FUNCTION_BLOCK sifb_bfb_inputs
  (* Standard: 61499-2 *)
  (* Version 0.1, 2018-00-07, hpea485, UOA *)
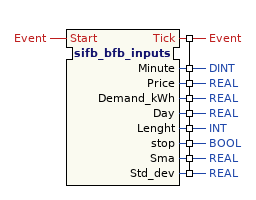
  EVENT_INPUT
    Start;
  END_EVENT
  EVENT_OUTPUT
    Tick WITH Minute, Price, Demand_kWh, Day, Lenght, stop, Sma, Std_dev;
  END_EVENT
  VAR_OUTPUT
    Minute : DINT;
    Price : REAL;
    Demand_kWh : REAL;
    Day : REAL;
    Lenght : INT;
    stop : BOOL;
    Sma : REAL;
    Std_dev : REAL;
  END_VAR
  VAR
    Var : DINT;
  END_VAR
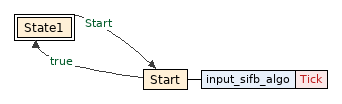
  EC_STATES
    State1;
    Start : input_sifb_algo -> Tick;
  END_STATES
  EC_TRANSITIONS
    Start TO State1 := true;
    State1 TO Start := Start;
  END_TRANSITIONS
  ALGORITHM input_sifb_algo IN C:
//#include "sifb_bfb_inputs.fb.Algorithm1.algo"
//#include "SMA_function.c"
#include <math.h>
static DINT current_minute = 0;
static DINT minute_for_demand = 0;
static DINT lol = 0;

static REAL Sma_tot = 0;
static int j = 1;
static REAL Std_dev;
static int nb_samples;

static int i = 0;
static int l = 8;
static int day = 0;
REAL Sma_forwrd=0;
REAL Sma_backwrd=0;
REAL Std_forwrd_sum = 0;
REAL Std_backwrd_sum = 0;
static bool stop = 0;
#define NUM_HALF_HOURS  48
#define NUM_DAYS        7 //31
me->stop = stop;



static REAL power_demand[1441][NUM_DAYS] = {
	{0,0,0,0,0,0,0},
	{176.7331, 236.0112, 169.5329, 136.7712, 100.643, 134.9339, 135.2902},
	{176.7331, 274.0112, 273.126, 280.6114, 275.0023, 273.324, 274.835},
	{176.7331, 274.0112, 273.126, 280.6114, 275.0023, 273.324, 274.835},
	{176.7331, 274.0112, 273.126, 280.6114, 275.0023, 273.324, 274.835},
	{176.7331, 274.0112, 273.126, 280.6114, 275.0023, 273.324, 274.835},
	{176.7331, 274.0112, 273.126, 280.6114, 275.0023, 273.324, 274.835},
	{176.7331, 274.0112, 273.126, 280.6114, 275.0023, 273.324, 274.835},
	{176.7331, 274.0112, 273.126, 280.6114, 275.0023, 273.324, 274.835},
	{176.7331, 274.0112, 273.126, 280.6114, 275.0023, 273.324, 274.835},
	{176.7331, 274.0112, 273.126, 280.6114, 275.0023, 273.324, 274.835},
	{176.7331, 274.0112, 273.126, 280.6114, 275.0023, 273.324, 274.835},
	{176.7331, 274.0112, 273.126, 280.6114, 275.0023, 273.324, 274.835},
	{176.7331, 274.0112, 273.126, 280.6114, 275.0023, 273.324, 274.835},
	{176.7331, 274.0112, 273.126, 280.6114, 275.0023, 273.324, 274.835},
	{176.7331, 274.0112, 273.126, 280.6114, 275.0023, 273.324, 274.835},
	{176.7331, 274.0112, 273.126, 280.6114, 275.0023, 273.324, 274.835},
	{176.7331, 274.0112, 273.126, 280.6114, 275.0023, 273.324, 274.835},
	{176.7331, 274.0112, 273.126, 280.6114, 275.0023, 273.324, 274.835},
	{176.7331, 274.0112, 273.126, 280.6114, 275.0023, 273.324, 274.835},
	{144.3122, 274.0112, 240.7051, 280.6114, 275.0023, 240.9031, 274.835},
	{144.3122, 209.1694, 240.7051, 280.6114, 242.5814, 240.9031, 242.4141},
	{144.3122, 209.1694, 240.7051, 280.6114, 242.5814, 208.4822, 242.4141},
	{144.3122, 209.1694, 240.7051, 280.6114, 242.5814, 208.4822, 242.4141},
	{144.3122, 175.2002, 240.7051, 212.673, 242.5814, 208.4822, 242.4141},
	{144.3122, 175.2002, 172.7667, 212.673, 208.6122, 208.4822, 174.4757},
	{110.343, 141.231, 138.7975, 212.673, 174.643, 174.513, 140.5065},
	{110.343, 106.231, 138.7975, 212.673, 174.643, 139.513, 140.5065},
	{132.634, 106.231, 103.7975, 142.673, 104.643, 104.513, 105.5065},
	{137.434, 106.231, 103.7975, 107.673, 104.643, 104.513, 105.5065},
	{207.2941, 106.231, 103.7975, 107.673, 104.643, 104.513, 105.5065},
	{207.2941, 106.231, 103.7975, 107.673, 104.643, 104.513, 105.5065},
	{207.2941, 106.231, 103.7975, 107.673, 104.643, 104.513, 105.5065},
	{207.2941, 106.231, 103.7975, 107.673, 104.643, 104.513, 105.5065},
	{207.2941, 106.231, 103.7975, 107.673, 104.643, 104.513, 105.5065},
	{207.2941, 106.231, 103.7975, 107.673, 104.643, 104.513, 105.5065},
	{207.2941, 106.231, 103.7975, 107.673, 103.313, 104.513, 105.5065},
	{202.4941, 106.231, 103.7975, 107.673, 135.7339, 104.513, 105.5065},
	{241.5941, 106.231, 103.7975, 107.673, 135.7339, 104.513, 105.5065},
	{241.5941, 106.231, 103.7975, 107.673, 135.7339, 104.513, 105.5065},
	{241.5941, 106.231, 137.4675, 107.673, 135.7339, 104.513, 105.5065},
	{241.5941, 106.231, 138.7975, 107.673, 135.7339, 136.9339, 105.5065},
	{241.5941, 106.231, 172.7667, 142.673, 135.7339, 136.9339, 105.5065},
	{241.5941, 106.231, 172.7667, 142.673, 135.7339, 136.9339, 105.5065},
	{241.5941, 106.231, 172.7667, 142.673, 135.7339, 136.9339, 105.5065},
	{241.5941, 106.231, 172.7667, 142.673, 135.7339, 136.9339, 105.5065},
	{241.5941, 106.231, 172.7667, 142.673, 135.7339, 136.9339, 105.5065},
	{241.5941, 104.901, 172.7667, 142.673, 135.7339, 136.9339, 105.5065},
	{241.5941, 104.901, 172.7667, 142.673, 135.7339, 136.9339, 105.5065},
	{241.5941, 104.901, 207.3659, 142.673, 135.7339, 136.9339, 105.5065},
	{209.1732, 104.901, 207.3659, 142.673, 135.7339, 136.9339, 105.5065},
	{209.1732, 104.901, 242.3659, 142.673, 135.7339, 136.9339, 105.5065},
	{209.1732, 104.901, 242.3659, 143.373, 135.7339, 136.9339, 105.5065},
	{209.1732, 104.901, 242.3659, 143.373, 135.7339, 136.9339, 139.8065},
	{209.1732, 137.3219, 242.3659, 143.373, 135.7339, 136.9339, 139.8065},
	{140.204, 137.3219, 242.3659, 143.373, 135.7339, 136.9339, 139.8065},
	{140.204, 137.3219, 242.3659, 143.373, 135.7339, 136.9339, 139.1065},
	{140.204, 137.3219, 242.3659, 177.3422, 103.313, 136.9339, 174.1065},
	{140.204, 136.6219, 242.3659, 177.3422, 103.313, 136.9339, 174.1065},
	{140.204, 171.6219, 242.3659, 177.3422, 103.313, 136.9339, 174.1065},
	{140.204, 171.6219, 242.3659, 177.3422, 103.313, 136.9339, 174.1065},
	{140.204, 172.9519, 242.3659, 177.3422, 103.313, 136.9339, 174.1065},
	{140.204, 172.9519, 208.3967, 177.3422, 103.313, 104.513, 174.1065},
	{105.204, 172.9519, 173.3967, 177.3422, 103.313, 140.143, 174.1065},
	{105.204, 207.2519, 173.3967, 177.3422, 137.9822, 140.143, 174.1065},
	{105.204, 207.2519, 173.3967, 142.3422, 104.013, 140.143, 174.1065},
	{105.204, 207.8819, 173.3967, 142.3422, 135.1039, 140.143, 174.1065},
	{105.204, 207.8819, 173.3967, 176.6422, 167.5248, 140.143, 174.1065},
	{105.204, 207.8819, 172.0667, 176.6422, 167.5248, 140.143, 174.1065},
	{105.204, 208.5819, 204.4876, 141.0122, 167.5248, 140.143, 174.1065},
	{105.204, 277.2203, 204.4876, 173.4331, 167.5248, 172.5639, 174.1065},
	{105.204, 277.2203, 170.5184, 173.4331, 167.5248, 172.5639, 174.1065},
	{105.204, 277.2203, 170.5184, 173.4331, 167.5248, 172.5639, 174.1065},
	{105.204, 244.7994, 170.5184, 173.4331, 167.5248, 172.5639, 172.7765},
	{105.204, 244.7994, 170.5184, 173.4331, 166.1948, 172.5639, 205.1974},
	{105.204, 244.7994, 170.5184, 173.4331, 198.6157, 172.5639, 205.1974},
	{105.204, 244.7994, 170.5184, 173.4331, 198.6157, 172.5639, 205.1974},
	{105.204, 244.7994, 204.8184, 173.4331, 198.6157, 172.5639, 205.1974},
	{140.5032, 244.7994, 169.8184, 173.7639, 198.6157, 172.5639, 205.1974},
	{140.5032, 244.7994, 169.8184, 138.1339, 198.6157, 172.5639, 170.1974},
	{140.5032, 244.7994, 169.8184, 170.5548, 198.6157, 204.3548, 135.1974},
	{140.5032, 244.7994, 169.8184, 170.5548, 198.6157, 171.9339, 135.1974},
	{140.5032, 244.7994, 169.8184, 170.5548, 198.6157, 204.3548, 170.8274},
	{140.5032, 244.7994, 169.8184, 205.5548, 198.6157, 204.3548, 135.1974},
	{140.5032, 209.7994, 169.8184, 205.5548, 167.5248, 204.3548, 167.6183},
	{140.5032, 209.7994, 169.8184, 205.5548, 135.1039, 205.0548, 167.6183},
	{141.2032, 209.7994, 137.3975, 205.5548, 135.1039, 237.694, 167.6183},
	{175.1724, 209.7994, 137.3975, 205.5548, 169.0731, 270.1149, 167.6183},
	{175.1724, 209.7994, 137.3975, 205.5548, 169.0731, 235.1149, 167.6183},
	{175.1724, 174.7994, 137.3975, 205.5548, 169.0731, 235.1149, 167.6183},
	{175.1724, 174.7994, 137.3975, 173.1339, 169.0731, 203.324, 167.6183},
	{175.1724, 106.861, 137.3975, 173.1339, 169.0731, 203.324, 167.6183},
	{175.1724, 106.861, 137.3975, 173.1339, 169.0731, 237.9932, 167.6183},
	{175.1724, 141.861, 137.3975, 173.1339, 137.3522, 237.9932, 135.1974},
	{175.1724, 141.861, 137.3975, 173.1339, 171.3214, 237.9932, 135.1974},
	{175.1724, 141.861, 137.3975, 173.1339, 171.3214, 237.9932, 135.1974},
	{175.1724, 141.861, 137.3975, 173.1339, 171.3214, 237.9932, 135.1974},
	{175.1724, 141.861, 137.3975, 173.1339, 171.3214, 237.9932, 135.1974},
	{175.1724, 141.861, 137.3975, 140.713, 171.3214, 237.9932, 135.1974},
	{175.1724, 141.861, 137.3975, 140.713, 171.3214, 237.9932, 135.1974},
	{175.1724, 141.861, 137.3975, 140.713, 171.3214, 237.9932, 134.5674},
	{171.7024, 141.861, 137.3975, 140.713, 171.3214, 237.9932, 166.9883},
	{171.7024, 175.8302, 102.3975, 140.713, 171.3214, 237.9932, 166.9883},
	{137.7332, 175.8302, 102.3975, 140.713, 171.3214, 205.5723, 166.9883},
	{137.7332, 208.2511, 102.3975, 140.713, 171.3214, 205.5723, 166.9883},
	{176.8332, 208.2511, 102.3975, 140.713, 171.3214, 173.1514, 134.5674},
	{176.8332, 208.2511, 102.3975, 140.713, 171.3214, 173.1514, 134.5674},
	{172.0332, 208.2511, 102.3975, 140.713, 171.3214, 173.1514, 134.5674},
	{176.1332, 208.2511, 102.3975, 140.713, 171.3214, 139.1822, 134.5674},
	{211.1332, 208.2511, 102.3975, 105.713, 171.3214, 139.1822, 134.5674},
	{246.1332, 208.2511, 102.3975, 105.713, 137.3522, 139.1822, 134.5674},
	{212.164, 208.2511, 102.3975, 105.713, 137.3522, 171.6031, 134.5674},
	{212.164, 208.2511, 136.3667, 106.343, 137.3522, 171.6031, 134.5674},
	{210.4785, 208.2511, 136.3667, 102.972, 135.6667, 169.9176, 134.5674},
	{210.4785, 208.2511, 100.712, 102.972, 101.6975, 169.9176, 134.5674},
	{210.4785, 208.2511, 134.6812, 102.342, 100.012, 169.9176, 132.8819},
	{208.793, 208.2511, 132.9957, 134.7629, 100.012, 134.2629, 132.8819},
	{205.422, 208.2511, 131.6647, 133.0774, 100.012, 164.8611, 131.1964},
	{203.7365, 206.5656, 166.6647, 129.7064, 100.012, 164.8611, 131.1964},
	{203.7365, 206.5656, 166.6647, 128.3764, 100.012, 164.8611, 131.1964},
	{203.7365, 206.5656, 166.6647, 128.3764, 100.012, 164.8611, 131.1964},
	{203.7365, 171.5656, 166.6647, 130.9164, 136.6512, 164.8611, 131.1964},
	{199.9765, 171.5656, 165.9647, 130.2864, 136.6512, 164.8611, 98.7755},
	{198.6465, 171.5656, 202.3047, 162.7073, 136.6512, 164.8611, 98.7755},
	{231.0674, 137.5964, 200.6192, 198.9673, 170.2649, 163.1756, 98.7755},
	{237.3674, 103.6755, 200.6192, 233.6365, 168.7649, 163.1756, 97.2755},
	{237.3674, 103.6755, 200.6192, 233.6365, 168.7649, 165.7156, 97.2755},
	{235.8674, 102.1755, 200.6192, 232.1365, 201.1858, 164.2156, 97.2755},
	{234.3674, 100.6755, 200.6192, 232.1365, 199.6858, 130.2947, 98.961},
	{234.3674, 99.1755, 200.6192, 232.1365, 167.2649, 130.2947, 97.461},
	{232.6819, 99.1755, 199.1192, 230.6365, 196.5003, 129.6492, 95.1455},
	{232.6819, 99.1755, 199.1192, 230.6365, 194.8148, 131.1492, 126.6964},
	{232.6819, 99.1755, 199.1192, 230.6365, 194.8148, 131.1492, 161.3656},
	{162.6819, 97.6755, 197.6192, 229.1365, 194.8148, 132.6492, 161.3656},
	{162.6819, 97.6755, 233.2492, 196.7156, 194.8148, 132.6492, 160.7356},
	{162.6819, 97.6755, 233.2492, 196.7156, 194.8148, 132.6492, 193.1565},
	{129.0219, 97.6755, 233.2492, 196.7156, 194.8148, 132.6492, 193.1565},
	{129.0219, 94.49, 233.2492, 193.5301, 194.8148, 133.9892, 228.4557},
	{129.0219, 94.49, 199.28, 193.5301, 194.8148, 136.5292, 228.4557},
	{125.2619, 94.49, 199.28, 193.5301, 194.1693, 136.5292, 228.4557},
	{129.0219, 94.49, 199.28, 193.5301, 194.1693, 102.56, 228.4557},
	{130.7074, 94.49, 199.28, 161.1092, 194.4693, 102.56, 228.4557},
	{98.2865, 97.03, 200.62, 161.1092, 194.4693, 136.5292, 228.4557},
	{98.2865, 97.73, 200.62, 159.6092, 160.5001, 136.5292, 228.4557},
	{96.7865, 131.6992, 199.12, 158.7392, 160.5001, 137.8592, 226.9557},
	{96.7865, 131.6992, 162.45, 158.1092, 160.5001, 137.8592, 226.9557},
	{91.9865, 131.3047, 159.8709, 156.5609, 160.5001, 137.8592, 225.9157},
	{95.7465, 133.4757, 161.5564, 159.4392, 126.5309, 136.5292, 227.6012},
	{97.432, 133.4757, 161.5564, 124.4392, 126.5309, 170.2901, 227.6012},
	{97.432, 167.4449, 161.5564, 125.7692, 93.71, 170.2901, 195.1803},
	{95.7465, 167.4449, 161.5564, 125.7692, 128.41, 168.9501, 230.8103},
	{89.4465, 167.4449, 161.5564, 125.7692, 128.41, 169.1356, 230.8103},
	{89.4465, 167.4449, 161.5564, 125.7692, 128.41, 169.1356, 230.8103},
	{94.5465, 166.4049, 196.2256, 124.7292, 128.41, 169.1356, 230.8103},
	{94.5465, 166.5904, 196.2256, 160.3839, 163.01, 167.6356, 195.3411},
	{94.5465, 201.8896, 196.2256, 160.6839, 164.6955, 167.6356, 195.3411},
	{94.5465, 201.8896, 161.5564, 160.6839, 164.6955, 203.2656, 162.9202},
	{94.5465, 201.8896, 196.5564, 163.4094, 164.6955, 203.2656, 196.8894},
	{94.5465, 201.8896, 196.5564, 164.9094, 165.8955, 203.2656, 196.8894},
	{95.2465, 201.8896, 161.5564, 164.9094, 165.8955, 203.9656, 164.2602},
	{125.4557, 201.8896, 161.5564, 164.9094, 168.4355, 237.2348, 164.2602},
	{120.6557, 201.2596, 163.2419, 164.9094, 168.4355, 238.2348, 198.5602},
	{121.4002, 233.6805, 163.2419, 166.2494, 169.7755, 238.2348, 198.5602},
	{151.4066, 233.6805, 163.2419, 166.2494, 169.7755, 238.2348, 198.5602},
	{155.5066, 233.6805, 130.821, 166.2494, 169.7755, 238.2348, 198.5602},
	{191.8466, 199.7113, 130.821, 167.5894, 169.7755, 237.1948, 198.5602},
	{195.6066, 199.7113, 130.821, 167.5894, 169.7755, 204.9111, 198.5602},
	{197.2921, 199.7113, 132.5065, 202.5894, 169.7755, 172.4902, 198.5602},
	{197.2921, 199.7113, 132.5065, 168.6202, 169.7755, 172.4902, 198.5602},
	{197.2921, 199.7113, 132.5065, 168.6202, 169.7755, 172.4902, 198.5602},
	{199.8321, 165.7421, 132.5065, 168.6202, 169.0755, 172.4902, 233.8594},
	{198.3321, 165.7421, 132.5065, 168.6202, 204.0755, 172.4902, 234.1594},
	{198.3321, 165.0421, 132.5065, 168.6202, 204.0755, 172.4902, 234.1594},
	{198.3321, 200.5421, 131.5065, 168.9602, 204.0755, 172.8302, 233.1594},
	{194.5721, 200.5421, 129.821, 169.9602, 169.0755, 172.8302, 233.1594},
	{194.5721, 200.5421, 197.5974, 169.9602, 169.0755, 172.8302, 235.6994},
	{198.3321, 200.5421, 162.2974, 135.991, 168.3755, 172.8302, 237.1994},
	{200.0176, 165.5729, 195.2666, 133.991, 166.7455, 172.8302, 200.8449},
	{200.0176, 165.5729, 195.2666, 133.991, 164.1664, 172.8302, 231.5803},
	{200.0176, 165.0729, 161.8457, 132.031, 161.1664, 171.8302, 232.2658},
	{200.0176, 165.3729, 159.2666, 164.4519, 161.1664, 136.8302, 232.2658},
	{200.0176, 165.3729, 158.2266, 196.1728, 161.1664, 136.8302, 233.7658},
	{200.0176, 165.3729, 159.9121, 230.842, 160.4664, 136.8302, 199.7966},
	{166.0484, 134.452, 159.9121, 232.342, 161.4664, 102.861, 199.7966},
	{133.6275, 134.452, 159.9121, 232.342, 161.4664, 103.561, 164.7966},
	{132.6275, 134.452, 159.9121, 232.6728, 161.5064, 136.5302, 163.7966},
	{132.6275, 134.452, 159.9121, 234.1728, 161.5064, 136.5302, 163.7966},
	{132.6275, 133.122, 159.9121, 234.1728, 161.8064, 135.8302, 164.4966},
	{132.6275, 166.8884, 159.9121, 234.1728, 161.8064, 170.8302, 165.9966},
	{132.6275, 166.8884, 159.9121, 234.1728, 161.8064, 170.8302, 165.9966},
	{92.8275, 166.8884, 191.703, 265.2637, 161.8064, 170.8302, 164.9966},
	{96.2975, 166.2429, 191.703, 197.8428, 197.4364, 170.8302, 164.9966},
	{128.7184, 167.7429, 191.703, 230.2637, 197.4364, 170.8302, 164.9966},
	{128.7184, 167.7429, 193.203, 230.9092, 197.4364, 170.8302, 129.6974},
	{128.7184, 167.7429, 161.4121, 230.9092, 197.4364, 170.8302, 129.6974},
	{127.6784, 167.4029, 196.4121, 229.2237, 197.4364, 170.8302, 129.6974},
	{130.0639, 167.4029, 196.4121, 230.9092, 197.4364, 170.8302, 98.6065},
	{131.5639, 168.4429, 196.4121, 230.9092, 165.0155, 170.8302, 132.5757},
	{131.5639, 134.9429, 196.4121, 230.9092, 130.0155, 170.8302, 132.5757},
	{133.2494, 133.9429, 195.4121, 230.9092, 130.0155, 170.8302, 132.5757},
	{132.2494, 165.3638, 162.9912, 166.0674, 130.0155, 169.8302, 132.5757},
	{167.2494, 168.5729, 165.982, 167.5674, 130.0155, 170.8302, 132.5757},
	{167.2494, 168.5729, 163.952, 165.0274, 130.0155, 169.8302, 132.5757},
	{167.2494, 169.5729, 195.7429, 166.7129, 130.0155, 170.8302, 166.8757},
	{167.2494, 169.2729, 228.1638, 166.7129, 130.0155, 170.8302, 166.8757},
	{163.1494, 170.7729, 228.8638, 166.7129, 130.0155, 170.8302, 166.8757},
	{167.9494, 170.7729, 230.3638, 166.7129, 130.0155, 136.861, 166.8757},
	{232.4178, 170.7729, 230.3638, 166.7129, 130.0155, 135.531, 166.8757},
	{236.5178, 138.352, 230.3638, 166.7129, 130.0155, 167.9519, 166.8757},
	{205.0969, 138.352, 229.3638, 166.7129, 130.0155, 166.6219, 165.8757},
	{205.0969, 138.352, 229.3638, 166.7129, 129.6855, 198.0028, 165.8757},
	{205.0969, 138.352, 229.3638, 166.7129, 161.1064, 199.6883, 165.8757},
	{205.0969, 138.352, 229.3638, 99.292, 162.1064, 199.6883, 165.8757},
	{205.0969, 173.6512, 228.3638, 98.292, 162.1064, 164.6883, 165.8757},
	{205.0969, 173.0212, 228.3638, 98.292, 162.1064, 164.6883, 165.8757},
	{205.0969, 207.3212, 228.3638, 98.292, 127.1064, 164.6883, 198.2966},
	{205.0969, 239.7421, 228.3638, 98.292, 127.1064, 164.6883, 165.8757},
	{205.0969, 205.4421, 228.3638, 98.292, 127.1064, 164.6883, 197.9566},
	{205.0969, 239.4113, 228.3638, 98.292, 127.1064, 199.9875, 165.6729},
	{205.0969, 239.4113, 228.3638, 98.292, 162.1064, 199.9875, 165.6729},
	{205.0969, 239.4113, 228.3638, 98.292, 162.1064, 199.9875, 165.6729},
	{205.0969, 239.4113, 163.1429, 98.292, 162.1064, 199.9875, 165.3329},
	{205.0969, 239.4113, 129.852, 99.622, 162.1064, 199.9875, 167.0184},
	{205.0969, 239.4113, 164.8212, 133.5912, 162.1064, 199.9875, 167.0184},
	{205.0969, 241.6113, 164.8212, 133.5912, 162.1064, 199.9875, 167.0184},
	{240.7269, 241.6113, 165.8212, 133.5912, 162.1064, 199.9875, 198.8093},
	{240.7269, 205.1113, 131.5212, 133.5912, 162.1064, 167.5666, 198.8093},
	{206.7577, 240.5805, 133.0212, 133.5912, 163.1064, 167.5666, 132.7184},
	{171.7577, 205.2813, 133.0212, 133.5912, 163.1064, 167.5666, 201.6876},
	{171.7577, 237.7022, 134.0212, 168.8904, 163.1064, 134.4457, 201.6876},
	{171.7577, 237.7022, 134.0212, 168.8904, 130.6855, 134.4457, 201.6876},
	{171.7577, 237.7022, 134.0212, 169.5204, 130.6855, 135.1457, 201.6876},
	{137.7885, 237.7022, 133.7212, 204.1896, 132.031, 169.1149, 202.3876},
	{137.7885, 237.7022, 135.2212, 205.1896, 130.6855, 169.1149, 203.8876},
	{137.7885, 205.2813, 135.2212, 205.1896, 131.6855, 168.7749, 203.8876},
	{132.9885, 205.2813, 135.2212, 205.1896, 131.6855, 170.4604, 203.8876},
	{172.0885, 171.3121, 135.2212, 205.1896, 131.6855, 170.4604, 171.4667},
	{170.7585, 171.3121, 135.2212, 205.1896, 131.6855, 170.4604, 171.4667},
	{203.1794, 171.3121, 135.9212, 205.1896, 131.6855, 170.4604, 171.4667},
	{203.1794, 171.3121, 137.4212, 205.1896, 131.6855, 136.4912, 171.4667},
	{203.1794, 137.3429, 137.4212, 205.1896, 131.6855, 136.4912, 171.1267},
	{203.1794, 137.3429, 137.4212, 205.1896, 131.6855, 136.4912, 172.8122},
	{203.1794, 137.3429, 137.4212, 205.1896, 131.6855, 137.1212, 172.8122},
	{203.1794, 137.3429, 137.4212, 205.1896, 96.6855, 137.1212, 172.8122},
	{203.1794, 137.3429, 137.4212, 204.8496, 96.6855, 137.1212, 172.8122},
	{203.1794, 136.6429, 137.4212, 206.5351, 96.6855, 137.1212, 174.1577},
	{203.1794, 136.6429, 169.8421, 172.5659, 96.6855, 137.1912, 174.1577},
	{203.1794, 136.0129, 169.8421, 172.5659, 96.0555, 204.5813, 174.1577},
	{203.1794, 136.0129, 135.8729, 172.5659, 128.4764, 204.2813, 174.1577},
	{203.1794, 136.0129, 135.8729, 172.5659, 129.4764, 205.7813, 138.843},
	{203.1794, 136.0129, 135.8729, 172.5659, 130.8219, 205.7813, 139.843},
	{203.1794, 136.0129, 138.0729, 172.5659, 129.1364, 205.7813, 139.843},
	{203.1794, 136.0129, 138.0729, 138.5967, 130.8219, 238.2022, 139.843},
	{166.4939, 136.0129, 138.0729, 138.5967, 165.4911, 238.2022, 104.843},
	{166.4939, 136.7129, 138.0729, 138.5967, 166.4911, 236.8722, 104.843},
	{166.4939, 138.2129, 138.7729, 138.5967, 165.1511, 202.903, 104.843},
	{164.9939, 138.2129, 170.5421, 140.7967, 131.5374, 201.403, 104.843},
	{132.573, 138.2129, 171.5421, 105.3275, 163.9583, 237.033, 103.1575},
	{132.573, 138.2129, 172.2421, 106.8275, 163.9583, 237.033, 103.1575},
	{132.573, 138.2129, 206.2113, 106.8275, 165.2883, 235.533, 101.472},
	{97.573, 138.2129, 206.2113, 106.8275, 165.2883, 235.193, 101.472},
	{97.573, 136.5274, 206.2113, 106.8275, 163.9583, 236.8785, 101.472},
	{132.573, 136.5274, 206.2113, 107.5275, 196.3792, 236.8785, 101.472},
	{132.573, 136.5274, 206.2113, 141.4967, 196.3792, 236.8785, 135.4412},
	{132.573, 134.8419, 206.2113, 141.4967, 196.3792, 236.8785, 135.4412},
	{164.103, 170.1411, 173.7904, 141.4967, 228.8001, 204.4576, 135.4412},
	{167.573, 170.1411, 207.7596, 175.4659, 228.8001, 204.4576, 135.4412},
	{202.1939, 170.1411, 207.7596, 175.4659, 228.8001, 170.4884, 135.4412},
	{203.8794, 173.3502, 170.7749, 175.4659, 196.3792, 170.4884, 170.4412},
	{203.8794, 173.3502, 203.1958, 175.4659, 196.3792, 170.4884, 170.4412},
	{203.8794, 173.3502, 203.1958, 175.4659, 196.3792, 170.4884, 206.0712},
	{236.3003, 173.0194, 203.1958, 173.9659, 196.3792, 138.0675, 206.0712},
	{236.3003, 173.0194, 203.1958, 205.0568, 196.3792, 136.8675, 206.0712},
	{236.3003, 173.0194, 203.1958, 205.0568, 196.3792, 136.8675, 206.0712},
	{232.9293, 173.0194, 203.1958, 205.0568, 196.3792, 169.3367, 206.0712},
	{232.9293, 173.0194, 203.1958, 205.0568, 196.3792, 167.6512, 206.0712},
	{232.9293, 173.0194, 203.1958, 205.0568, 163.9583, 167.6512, 206.0712},
	{232.9293, 171.9639, 169.2266, 173.2659, 163.9583, 167.6512, 206.0712},
	{232.9293, 206.2639, 169.2266, 208.2659, 163.9583, 167.6512, 206.0712},
	{232.9293, 171.9794, 169.2266, 208.2659, 163.9583, 167.6512, 206.0712},
	{232.9293, 239.4003, 169.2266, 208.2659, 163.9583, 167.6512, 207.4167},
	{232.9293, 238.7548, 169.2266, 208.2659, 131.5374, 165.9657, 206.7712},
	{232.9293, 242.7948, 132.9419, 208.2659, 131.5374, 129.4657, 208.2712},
	{232.9293, 274.5857, 165.3628, 206.5804, 131.5374, 128.4257, 208.2712},
	{232.9293, 242.1648, 165.3628, 173.3112, 131.5374, 130.1112, 208.2712},
	{232.9293, 274.5857, 167.0483, 205.5949, 135.1157, 131.7967, 208.2712},
	{199.5229, 274.5857, 202.6783, 171.6257, 169.0849, 131.7967, 209.3267},
	{233.4921, 240.6165, 202.3475, 171.6257, 169.0849, 131.7967, 241.7476},
	{198.4921, 240.6165, 169.9266, 171.6257, 169.0849, 166.0967, 207.7784},
	{166.0712, 240.6165, 169.9266, 170.5857, 165.8994, 166.0967, 207.7784},
	{131.0712, 240.6165, 169.9266, 172.2712, 165.8994, 166.0967, 207.7784},
	{131.0712, 240.6165, 169.9266, 170.7712, 165.8994, 166.0967, 207.7784},
	{124.5857, 238.931, 169.9266, 170.7712, 165.8994, 165.3967, 207.7784},
	{123.0857, 238.931, 169.9266, 170.7712, 165.8994, 166.3967, 172.7784},
	{123.0857, 238.931, 172.4666, 170.7712, 165.8994, 166.3967, 137.7784},
	{162.4757, 238.931, 168.2411, 170.7712, 164.3994, 166.3967, 137.7784},
	{164.1612, 204.9618, 168.9266, 170.7712, 164.3994, 166.3967, 137.7784},
	{164.1612, 172.5409, 168.9266, 235.8313, 199.6986, 166.3967, 137.7784},
	{164.1612, 172.5409, 168.9266, 235.8313, 199.6986, 166.3967, 137.7784},
	{164.1612, 172.5409, 168.9266, 235.8313, 199.6986, 132.4275, 137.7784},
	{164.1612, 172.5409, 136.5057, 203.4104, 199.6986, 132.4275, 137.7784},
	{164.1612, 172.5409, 136.5057, 204.9104, 199.6986, 166.7275, 137.7784},
	{164.1612, 140.12, 136.5057, 205.5404, 198.1986, 166.7275, 137.7784},
	{164.1612, 106.8055, 170.8057, 205.5404, 198.1986, 166.7275, 137.7784},
	{164.1612, 105.12, 169.8057, 205.5404, 198.1986, 166.7275, 103.8575},
	{165.8467, 141.1055, 169.8057, 205.5404, 198.1986, 169.2675, 138.1575},
	{165.8467, 139.6055, 169.8057, 205.5404, 164.2294, 204.5667, 138.1575},
	{165.8467, 139.6055, 169.8057, 171.5712, 130.2602, 204.5667, 139.4975},
	{164.1612, 139.6055, 169.8057, 171.5712, 130.2602, 204.5667, 139.4975},
	{164.1612, 140.9455, 169.8057, 171.5712, 130.2602, 204.5667, 137.812},
	{130.192, 140.9455, 135.8365, 206.5712, 129.2602, 204.5667, 170.2812},
	{125.392, 140.9455, 135.8365, 206.5712, 129.2602, 204.5667, 170.2812},
	{125.392, 140.2455, 135.8365, 206.5712, 129.2602, 205.1967, 205.9112},
	{125.392, 140.9455, 135.8365, 206.5712, 129.2602, 205.1967, 205.5804},
	{129.492, 174.9147, 135.8365, 206.5712, 163.5602, 204.1967, 205.5804},
	{129.492, 174.2847, 135.8365, 206.5712, 163.5602, 204.1967, 205.5804},
	{128.162, 206.7056, 135.8365, 206.5712, 163.5602, 203.4967, 205.5804},
	{160.5829, 206.7056, 135.8365, 206.5712, 163.5602, 204.4967, 205.5804},
	{160.5829, 206.7056, 135.8365, 206.5712, 164.8902, 204.4967, 205.5804},
	{121.8229, 206.7056, 134.151, 203.3857, 163.5602, 204.4967, 205.5804},
	{129.8084, 206.7056, 134.151, 203.3857, 195.9811, 204.4967, 205.5804},
	{129.8084, 205.7056, 134.151, 203.7165, 195.9811, 204.4967, 205.5804},
	{129.8084, 204.2056, 134.151, 169.4165, 195.9811, 204.4967, 204.0804},
	{129.8084, 202.7056, 134.151, 203.3857, 195.9811, 204.4967, 202.5804},
	{129.8084, 202.7056, 134.151, 203.3857, 195.9811, 204.4967, 202.5804},
	{129.8084, 202.7056, 134.151, 203.3857, 195.9811, 204.4967, 202.5804},
	{129.8084, 202.7056, 169.4502, 203.3857, 195.9811, 169.4967, 202.5804},
	{129.8084, 202.7056, 168.1202, 203.3857, 228.402, 169.4967, 202.5804},
	{129.8084, 170.2456, 169.4502, 168.3857, 228.402, 135.5275, 202.5804},
	{125.7084, 168.7456, 202.4194, 169.8857, 228.402, 135.5275, 202.5804},
	{128.8229, 168.7456, 201.3886, 169.8857, 228.402, 133.842, 202.5804},
	{162.7921, 168.7456, 201.3886, 169.8857, 228.402, 134.542, 166.9257},
	{159.0321, 163.9456, 201.7194, 168.2002, 228.402, 168.5112, 131.9257},
	{165.3321, 168.7456, 200.2194, 168.2002, 227.402, 169.8512, 131.9257},
	{165.3321, 167.5456, 200.2194, 166.7002, 227.742, 171.3512, 131.9257},
	{165.3321, 167.5456, 200.2194, 166.7002, 227.742, 172.5512, 131.9257},
	{165.3321, 135.1247, 200.2194, 165.6694, 227.042, 172.5512, 131.9257},
	{132.9112, 101.1555, 200.2194, 131.9102, 228.042, 136.5512, 97.9565},
	{128.8112, 101.1555, 200.2194, 161.7911, 193.042, 136.5512, 97.9565},
	{132.5712, 102.6555, 202.4194, 162.4766, 160.6211, 136.5512, 97.3265},
	{134.2567, 102.6555, 202.4194, 162.4766, 160.6211, 136.5512, 129.7474},
	{132.7567, 102.6555, 202.4194, 162.4766, 126.6519, 136.5512, 131.4329},
	{132.7567, 101.1555, 202.4194, 162.4766, 128.1519, 137.5512, 131.4329},
	{132.7567, 102.6555, 200.9194, 162.4766, 128.1519, 136.5512, 131.4329},
	{129.6967, 102.6555, 202.4194, 162.4766, 128.1519, 137.5512, 131.4329},
	{167.4259, 101.6155, 202.4194, 198.4166, 128.1519, 136.5512, 130.7329},
	{169.1114, 103.301, 234.8403, 164.1474, 128.1519, 136.5512, 130.4029},
	{204.4106, 103.301, 200.8711, 129.8474, 128.1519, 136.5512, 162.8238},
	{206.9506, 103.301, 200.8711, 167.0021, 95.731, 136.5512, 161.8238},
	{206.9506, 103.301, 200.8711, 167.0021, 94.691, 134.8657, 161.8238},
	{206.9506, 102.261, 200.8711, 167.0021, 96.3765, 134.8657, 161.8238},
	{206.9506, 103.9465, 166.9019, 167.0021, 96.3765, 134.2357, 161.8238},
	{172.9814, 103.9465, 166.9019, 167.0021, 96.3765, 134.2357, 161.8238},
	{172.9814, 102.4465, 166.9019, 167.0021, 96.3765, 134.2357, 160.1383},
	{207.9814, 172.7457, 165.4019, 167.0021, 95.6765, 134.8657, 194.8075},
	{207.9814, 205.1666, 130.4019, 167.0021, 95.0465, 170.5657, 160.8383},
	{207.9814, 205.1666, 132.0874, 167.0021, 127.4674, 170.5657, 194.8075},
	{206.9814, 205.1666, 133.4329, 167.0021, 127.4674, 170.5657, 194.8075},
	{206.9814, 205.1666, 132.0874, 167.0021, 126.4674, 170.5657, 194.8075},
	{206.9814, 203.6666, 132.7474, 133.5812, 126.4674, 170.5657, 199.8875},
	{201.8814, 203.6666, 134.4329, 131.8957, 126.4674, 170.5657, 164.9266},
	{201.8814, 202.9666, 136.1184, 131.8957, 126.4674, 170.5657, 165.5721},
	{205.9814, 203.9666, 132.9329, 131.8957, 126.4674, 170.5657, 166.6121},
	{206.9814, 203.9666, 133.1184, 132.5957, 126.4674, 170.5657, 166.0866},
	{206.9814, 203.9666, 133.1184, 134.0957, 127.1674, 172.2512, 169.2721},
	{206.9814, 202.9666, 100.6975, 134.0957, 130.8674, 172.2512, 136.8512},
	{206.9814, 202.9666, 100.9975, 134.0957, 130.8674, 171.9057, 169.2721},
	{173.0122, 202.9666, 99.4975, 134.0957, 129.3674, 171.9057, 166.7321},
	{139.043, 202.9666, 99.4975, 134.0957, 130.8674, 171.9057, 169.9176},
	{139.043, 202.9666, 99.4975, 134.0957, 130.8674, 174.1057, 169.9176},
	{139.043, 202.9666, 99.4975, 134.0957, 130.8674, 171.5657, 169.9176},
	{139.043, 202.9666, 99.4975, 101.1265, 130.8674, 173.2512, 169.9176},
	{139.043, 202.9666, 99.4975, 101.1265, 131.4974, 173.2512, 169.9176},
	{134.943, 170.5457, 99.4975, 101.8265, 132.1974, 172.2512, 204.5868},
	{138.703, 170.5457, 99.4975, 135.1657, 133.7457, 172.2512, 204.5868},
	{140.3885, 170.5457, 99.4975, 167.5866, 132.0602, 172.2512, 168.9176},
	{140.3885, 136.5765, 100.1975, 167.5866, 132.0602, 172.2512, 203.9176},
	{140.3885, 136.5765, 134.1667, 168.2266, 132.0602, 136.782, 237.8868},
	{140.3885, 136.5765, 134.1667, 168.2266, 132.0602, 171.082, 237.8868},
	{140.3885, 135.5457, 134.1667, 168.2266, 130.7302, 171.082, 203.9176},
	{140.3885, 135.5457, 134.1667, 169.5666, 163.1511, 171.082, 202.4176},
	{105.3885, 135.5457, 134.3367, 168.9266, 163.1511, 135.0965, 202.4176},
	{105.3885, 134.8457, 168.4667, 204.5813, 162.8111, 169.0657, 202.4176},
	{105.3885, 135.8457, 203.4359, 204.5813, 198.7958, 169.0657, 202.4176},
	{105.3885, 135.8457, 203.4359, 204.5813, 198.7958, 169.0812, 202.4176},
	{99.943, 135.8457, 203.4359, 204.5813, 198.7958, 170.4112, 202.4176},
	{136.1239, 166.9366, 203.4359, 204.5813, 198.7958, 203.7349, 170.2967},
	{137.8094, 134.2757, 203.4359, 204.5813, 198.4503, 205.2349, 170.2967},
	{137.8094, 204.6449, 203.4359, 204.5813, 198.4503, 205.2349, 205.5959},
	{136.8094, 207.1449, 201.6959, 204.5813, 198.6503, 205.2349, 205.5959},
	{132.0094, 206.8449, 238.3814, 204.5813, 198.6503, 203.9049, 205.5959},
	{135.4794, 208.3449, 238.3814, 204.5813, 198.6503, 236.3258, 205.5959},
	{167.9003, 208.3449, 238.3814, 204.5813, 198.6503, 235.6258, 205.5959},
	{167.9003, 209.8449, 238.3814, 171.8204, 198.3103, 235.6258, 208.1359},
	{167.9003, 209.8449, 238.3814, 173.5059, 199.9958, 236.3258, 208.1359},
	{167.9003, 209.8449, 238.3814, 173.5059, 200.6958, 237.8258, 208.1359},
	{167.9003, 209.8449, 238.3814, 139.5367, 236.0105, 237.8258, 208.1359},
	{167.9003, 209.8449, 204.4122, 139.5367, 271.6405, 237.8258, 208.1359},
	{163.1003, 209.8449, 204.4122, 139.5367, 239.2196, 237.8258, 208.1359},
	{167.9003, 209.8449, 203.7122, 139.5367, 204.2504, 237.1958, 174.1667},
	{169.4003, 175.8757, 204.7122, 139.5367, 203.6049, 269.6167, 139.1667},
	{169.4003, 175.8757, 204.7122, 139.5367, 205.1049, 269.6167, 139.1667},
	{169.4003, 175.8757, 204.7122, 139.5367, 206.7904, 269.6167, 139.1667},
	{169.4003, 176.5757, 203.7122, 139.5367, 206.7904, 235.6475, 139.1667},
	{169.4003, 175.2457, 203.7122, 139.5367, 205.1049, 234.6167, 137.6667},
	{132.1794, 241.6358, 169.743, 139.5367, 206.7904, 234.6167, 137.6667},
	{132.1794, 242.2813, 169.743, 105.5675, 172.8212, 234.6167, 137.6667},
	{132.1794, 240.7813, 169.743, 105.5675, 171.4912, 234.6167, 137.6667},
	{133.9639, 239.0958, 134.743, 105.5675, 203.9121, 200.6475, 137.6667},
	{164.8848, 206.1666, 134.743, 104.3675, 203.9121, 200.6475, 136.9667},
	{164.8848, 242.9658, 134.743, 104.3675, 203.9121, 168.2266, 102.9975},
	{132.4639, 242.9658, 134.743, 104.3675, 205.2576, 168.2266, 101.312},
	{132.4639, 242.9658, 134.743, 103.0275, 205.2576, 168.2266, 136.6112},
	{127.6639, 242.9658, 134.743, 104.713, 203.5721, 168.2266, 136.3367},
	{127.6639, 242.9658, 134.743, 140.343, 205.2576, 168.2266, 202.033},
	{127.6639, 207.9658, 99.743, 139.643, 205.2576, 168.2266, 202.033},
	{127.6639, 207.9658, 99.743, 139.013, 204.2576, 166.5411, 202.033},
	{132.4639, 207.9658, 99.3975, 171.4339, 170.2884, 166.5411, 202.033},
	{166.4331, 207.9658, 97.712, 170.4339, 170.2884, 134.1202, 204.233},
	{166.4331, 206.4658, 97.712, 205.7331, 170.2884, 132.4347, 202.733},
	{166.4331, 206.4658, 97.712, 205.7331, 135.2884, 132.0947, 204.233},
	{164.7476, 206.4658, 97.712, 205.7331, 135.2884, 133.7802, 204.233},
	{164.7476, 206.4658, 97.712, 205.7331, 135.2884, 133.7802, 204.233},
	{164.7476, 174.0449, 132.642, 202.9031, 135.2884, 133.7802, 205.733},
	{164.7476, 206.4658, 133.342, 235.324, 136.2884, 133.7802, 205.733},
	{164.7476, 206.4658, 167.3112, 235.324, 134.9484, 169.4102, 205.733},
	{164.7476, 206.4658, 167.3112, 235.324, 136.6339, 135.441, 205.733},
	{160.9876, 172.4966, 168.8112, 233.6385, 167.7248, 135.441, 205.733},
	{131.3967, 172.4966, 167.3112, 233.6385, 104.213, 135.441, 240.733},
	{134.8667, 172.4966, 168.8112, 233.6385, 138.1822, 135.441, 205.733},
	{163.1876, 172.4966, 168.8112, 233.6385, 172.1514, 135.441, 240.733},
	{163.1876, 138.5274, 168.8112, 233.6385, 172.1514, 133.941, 240.733},
	{159.4276, 136.8419, 168.8112, 233.6385, 172.1514, 133.941, 207.3121},
	{165.7276, 136.8419, 168.8112, 233.6385, 172.1514, 133.941, 207.3121},
	{165.7276, 136.8419, 168.8112, 233.6385, 172.1514, 135.6265, 207.3121},
	{165.7276, 136.8419, 168.8112, 201.2176, 172.1514, 136.3265, 174.8912},
	{169.8276, 136.8419, 168.8112, 201.2176, 172.1514, 170.2957, 175.222},
	{204.8276, 136.8419, 168.8112, 166.2176, 172.1514, 170.2957, 175.222},
	{204.8276, 136.8419, 167.8112, 166.2176, 172.1514, 170.2957, 175.222},
	{204.8276, 136.8419, 167.8112, 166.2176, 172.8514, 170.2957, 173.892},
	{206.3276, 136.8419, 167.8112, 166.2176, 174.3514, 170.5957, 206.3129},
	{170.6729, 136.8419, 167.8112, 166.5176, 174.3514, 170.5957, 206.3129},
	{205.9721, 135.8019, 167.8112, 132.5484, 174.3514, 171.4502, 206.3129},
	{205.9721, 137.4874, 167.8112, 100.1275, 174.3514, 171.4502, 206.3129},
	{206.6721, 105.0665, 167.8112, 99.4275, 174.3514, 171.4502, 206.3129},
	{208.1721, 105.0665, 167.8112, 134.4275, 174.3514, 171.4502, 207.6429},
	{208.1721, 105.0665, 132.8112, 133.7275, 173.3514, 171.4502, 206.3129},
	{208.1721, 105.0665, 132.8112, 168.7275, 173.3514, 171.4502, 238.7338},
	{208.1721, 105.0665, 132.8112, 168.7275, 173.3514, 171.4502, 238.7338},
	{172.2812, 105.0665, 132.8112, 168.7275, 173.3514, 171.4502, 238.7338},
	{172.2812, 105.0665, 133.142, 168.7275, 173.3514, 171.4502, 238.7338},
	{170.7812, 105.0665, 133.142, 168.7275, 173.3514, 171.4502, 238.7338},
	{204.7504, 139.0357, 134.8275, 168.7275, 139.3822, 136.4502, 238.7338},
	{243.8504, 139.0357, 134.8275, 167.042, 105.413, 136.4502, 238.7338},
	{243.8504, 173.0049, 134.8275, 167.042, 105.413, 136.4502, 238.7338},
	{243.8504, 137.7057, 134.8275, 167.042, 105.413, 136.4502, 238.7338},
	{243.8504, 205.7566, 134.8275, 167.042, 105.413, 170.4194, 203.7338},
	{243.8504, 205.7566, 134.8275, 167.042, 105.413, 171.7494, 203.7338},
	{243.8504, 206.4566, 134.8275, 167.042, 105.413, 172.1049, 171.3129},
	{243.8504, 240.4258, 168.7967, 167.042, 105.413, 202.8403, 171.3129},
	{243.8504, 240.4258, 168.7967, 167.042, 105.413, 170.7421, 171.3129},
	{243.8504, 239.7258, 133.4975, 167.042, 105.413, 203.0258, 136.3129},
	{243.8504, 274.695, 165.9184, 167.042, 105.413, 204.7113, 136.3129},
	{207.1649, 273.0095, 165.9184, 202.672, 140.7122, 204.7113, 136.3129},
	{207.1649, 273.0095, 165.9184, 202.672, 140.7122, 203.7113, 136.3129},
	{207.1649, 273.0095, 165.9184, 202.672, 140.7122, 203.7113, 103.892},
	{207.1649, 273.0095, 165.9184, 202.672, 140.7122, 203.7113, 103.892},
	{207.4957, 273.0095, 165.9184, 202.672, 140.7122, 203.7113, 103.892},
	{207.4957, 273.0095, 165.9184, 202.672, 140.7122, 203.7113, 103.892},
	{205.8102, 273.0095, 200.9184, 202.672, 140.7122, 204.7113, 103.892},
	{207.4957, 273.0095, 200.9184, 166.172, 140.7122, 204.7113, 102.2065},
	{207.4957, 273.0095, 200.9184, 131.172, 140.7122, 205.4113, 102.2065},
	{207.4957, 273.0095, 199.2329, 131.172, 141.3422, 239.3805, 102.2065},
	{207.4957, 273.0095, 164.2329, 132.8575, 141.3422, 239.3805, 102.2065},
	{204.4474, 239.0403, 164.2329, 131.172, 141.3422, 239.3805, 102.2065},
	{204.4474, 239.0403, 162.5474, 131.172, 176.0114, 239.3805, 102.2065},
	{204.4474, 206.6194, 162.5474, 131.172, 211.0114, 239.3805, 102.2065},
	{204.4474, 206.6194, 162.5474, 131.172, 211.0114, 207.2904, 137.5057},
	{204.4474, 206.6194, 162.5474, 131.172, 211.0114, 207.2904, 137.5057},
	{169.4474, 203.4339, 197.2166, 131.172, 211.0114, 205.7904, 137.5057},
	{169.4474, 205.1194, 161.9174, 131.172, 209.3259, 204.7904, 137.5057},
	{165.3474, 204.7739, 194.3383, 129.672, 209.3259, 204.7904, 137.5057},
	{167.8874, 170.1047, 161.9174, 129.672, 209.3259, 238.7596, 137.5057},
	{171.3574, 170.1047, 161.9174, 162.0929, 209.3259, 204.4596, 135.8202},
	{203.7783, 136.1355, 161.9174, 162.0929, 209.3259, 204.4596, 135.8202},
	{203.7783, 136.1355, 161.9174, 162.0929, 209.3259, 204.4596, 134.1347},
	{203.7783, 136.1355, 161.9174, 162.0929, 209.3259, 169.1604, 169.7647},
	{198.9783, 134.6355, 161.9174, 162.0929, 209.3259, 201.5813, 169.7647},
	{202.4483, 134.6355, 161.9174, 162.0929, 208.1567, 201.5813, 169.7647},
	{234.8692, 134.6355, 162.9174, 127.0929, 173.1567, 201.5813, 169.5947},
	{195.0692, 134.6355, 162.9174, 162.0929, 206.6567, 201.5813, 169.5947},
	{195.0692, 134.6355, 162.9174, 163.7784, 206.6567, 201.5813, 167.9092},
	{160.9628, 133.6355, 159.7319, 160.5929, 206.6567, 201.5813, 169.1192},
	{161.9628, 133.6355, 159.4319, 162.2784, 206.6567, 201.5813, 201.5401},
	{161.9628, 133.6355, 125.9319, 162.2784, 206.6567, 201.5813, 201.5401},
	{166.7628, 133.6355, 125.9319, 162.2784, 172.6875, 168.6121, 202.8856},
	{200.732, 133.6355, 157.7228, 162.2784, 172.6875, 168.6121, 201.5401},
	{200.102, 133.6355, 190.1437, 161.9384, 172.6875, 168.6121, 202.5401},
	{231.5229, 133.6355, 190.1437, 163.6239, 172.6875, 168.6121, 168.5709},
	{231.5229, 164.7264, 159.0528, 163.6239, 172.6875, 167.6121, 168.5709},
	{230.0229, 166.9047, 193.022, 163.6239, 172.6875, 167.6121, 168.5709},
	{230.0229, 202.2355, 193.3528, 195.4148, 172.6875, 165.9266, 168.5709},
	{230.0229, 202.2355, 193.3528, 162.9939, 172.6875, 165.9266, 168.5709},
	{230.0229, 202.2355, 157.7228, 130.573, 137.6875, 165.9266, 170.0709},
	{197.602, 202.2355, 190.1437, 162.9939, 137.6875, 165.9266, 167.0709},
	{195.5765, 202.2355, 190.1437, 162.9939, 172.6875, 130.6274, 168.5709},
	{197.262, 202.2355, 190.1437, 162.8084, 172.6875, 164.5483, 168.5709},
	{193.502, 167.2355, 189.8037, 195.2293, 171.1875, 164.5483, 203.5709},
	{193.502, 167.5355, 191.4892, 195.2293, 205.1567, 166.7174, 203.5709},
	{199.802, 167.5355, 191.4892, 227.0202, 206.5022, 168.4029, 238.5709},
	{167.3811, 166.4955, 191.4892, 197.6148, 204.8167, 202.5329, 238.5709},
	{167.3811, 168.181, 194.0292, 231.584, 205.1722, 202.5329, 171.15},
	{167.3811, 168.181, 194.0292, 231.584, 237.5931, 236.5021, 171.15},
	{167.3811, 168.181, 194.0292, 231.584, 237.5931, 236.5021, 171.15},
	{167.3811, 168.181, 194.7292, 196.584, 237.5931, 236.5021, 173.69},
	{167.6811, 168.181, 196.2775, 194.8985, 235.9076, 236.5021, 172.19},
	{167.6811, 168.181, 163.8566, 194.8985, 235.9076, 236.5021, 172.19},
	{135.2602, 168.181, 163.8566, 194.8985, 200.9076, 236.5021, 203.2809},
	{135.2602, 166.681, 163.8566, 194.8985, 200.9076, 236.5021, 201.9409},
	{135.2602, 166.681, 162.5111, 194.8985, 200.9076, 236.5021, 172.5355},
	{102.9765, 169.221, 163.5111, 194.8985, 200.9076, 236.5021, 206.5047},
	{135.3974, 165.181, 163.5111, 194.8985, 200.9076, 236.5021, 205.5047},
	{135.3974, 165.3665, 131.0902, 194.8985, 200.9076, 236.5021, 205.8047},
	{135.3974, 167.052, 131.0902, 197.044, 200.9076, 236.5021, 205.8047},
	{133.8974, 132.052, 132.7757, 164.6231, 199.9076, 236.5021, 204.3047},
	{133.1974, 97.052, 132.7757, 163.2776, 199.9076, 236.5021, 204.3047},
	{134.1974, 128.4729, 132.7757, 164.2776, 199.9076, 236.5021, 204.3047},
	{134.1974, 128.4729, 132.7757, 164.2776, 199.9076, 204.0812, 205.8047},
	{134.1974, 128.4729, 132.7757, 131.8567, 164.9076, 204.0812, 205.8047},
	{169.8274, 128.4729, 132.7757, 131.8567, 97.0175, 204.0812, 208.3447},
	{169.8274, 128.4729, 132.7757, 134.3967, 96.3175, 204.0812, 174.6847},
	{169.8274, 128.4729, 132.7757, 134.3967, 93.292, 204.0812, 172.1447},
	{169.8274, 128.4729, 132.7757, 134.3967, 96.4775, 204.0812, 175.0302},
	{169.8274, 128.4729, 132.7757, 100.5675, 96.4775, 134.0812, 140.0302},
	{169.8274, 128.4729, 168.4057, 100.5675, 96.4775, 134.0812, 140.7302},
	{169.8274, 127.4329, 168.4057, 100.5675, 96.4775, 134.0812, 174.6994},
	{169.8274, 128.0784, 168.4057, 135.5675, 96.4775, 100.112, 174.6994},
	{169.8274, 129.7639, 167.7757, 100.2675, 93.9375, 100.742, 174.6994},
	{169.8274, 129.7639, 201.6966, 166.6576, 97.123, 133.542, 174.6994},
	{136.4065, 129.1339, 201.6966, 166.6576, 97.123, 170.042, 174.6994},
	{136.4065, 161.5548, 167.7274, 164.9721, 94.1075, 170.042, 174.6994},
	{132.9365, 161.5548, 167.7274, 164.9721, 94.1075, 170.042, 140.7302},
	{171.7057, 161.5548, 167.7274, 164.9721, 93.9475, 170.042, 140.0302},
	{171.7057, 161.5548, 167.7274, 164.9721, 126.3684, 170.042, 140.0302},
	{171.7057, 161.5548, 167.7274, 164.9721, 126.3684, 170.042, 140.0302},
	{171.7057, 161.5548, 203.3574, 164.9721, 127.0684, 170.042, 140.0302},
	{171.7057, 129.1339, 203.3574, 163.9721, 161.0376, 169.042, 140.7302},
	{171.7057, 129.1339, 203.3574, 163.9721, 161.0376, 167.3565, 142.2302},
	{171.7057, 129.1339, 203.3574, 163.9721, 161.0376, 167.3565, 142.2302},
	{171.7057, 129.1339, 203.3574, 197.9413, 161.0376, 169.042, 142.2302},
	{171.7057, 128.1339, 203.3574, 198.6413, 161.0376, 167.3565, 142.2302},
	{171.7057, 128.1339, 203.3574, 232.6105, 161.0376, 169.042, 142.2302},
	{171.7057, 128.1339, 202.3574, 232.6105, 161.0376, 169.042, 142.2302},
	{167.9457, 161.3031, 202.3574, 231.6105, 161.0376, 200.8329, 142.2302},
	{134.5757, 161.9331, 202.3574, 231.6105, 161.0376, 168.412, 142.2302},
	{138.0457, 196.9331, 202.3574, 231.6105, 161.0376, 200.8329, 142.2302},
	{170.4666, 195.2476, 170.5665, 232.2405, 161.0376, 200.8329, 108.261},
	{170.4666, 195.2476, 170.5665, 232.2405, 161.0376, 199.8329, 140.7302},
	{170.4666, 162.8267, 170.5665, 234.8196, 161.0376, 200.4784, 140.7302},
	{170.4666, 162.8267, 170.5665, 198.1896, 161.0376, 199.1329, 140.7302},
	{170.4666, 162.8267, 170.5665, 230.6105, 161.0376, 200.1329, 139.2302},
	{170.4666, 162.8267, 170.5665, 196.6413, 161.0376, 200.1329, 174.5294},
	{170.4666, 162.5267, 170.5665, 197.9868, 161.0376, 165.1329, 174.5294},
	{170.4666, 196.4959, 170.5665, 196.3013, 161.0376, 130.1329, 174.5294},
	{170.4666, 196.4959, 170.5665, 197.9868, 161.0376, 130.1329, 174.5294},
	{168.9666, 198.1814, 170.5665, 197.9868, 161.0376, 130.1329, 174.5294},
	{168.9666, 198.1814, 169.0665, 197.9868, 161.0376, 130.8329, 173.0294},
	{134.9974, 199.3414, 168.721, 197.9868, 127.0684, 164.8021, 173.0294},
	{130.1974, 201.0269, 202.6902, 197.9868, 125.5684, 164.8021, 173.0294},
	{133.6674, 198.4869, 168.8902, 197.9868, 124.2384, 164.8021, 174.0294},
	{166.0883, 201.1724, 167.8902, 197.9868, 156.6593, 165.8021, 175.5294},
	{166.0883, 200.1724, 167.8902, 164.0176, 156.6593, 165.1721, 177.0294},
	{161.2883, 201.1724, 168.2302, 164.0176, 156.6593, 197.593, 177.0294},
	{201.3875, 201.1724, 168.2302, 130.0484, 157.3593, 163.4866, 175.8294},
	{229.7567, 201.1724, 168.2302, 130.0484, 158.8593, 163.4866, 175.8294},
	{234.5567, 167.2032, 168.2302, 130.3884, 158.8593, 163.4866, 175.8294},
	{234.605, 167.2032, 202.8602, 130.3884, 158.8593, 163.4866, 175.8294},
	{233.105, 167.2032, 202.8602, 132.5884, 128.1239, 161.9866, 175.8294},
	{233.105, 167.2032, 202.8602, 132.5884, 128.1239, 161.9866, 175.8294},
	{233.105, 167.2032, 202.8602, 132.5884, 129.6239, 161.9866, 141.8602},
	{233.105, 167.2032, 202.8602, 100.1675, 162.0839, 197.2858, 175.8294},
	{233.105, 167.2032, 202.8602, 100.1675, 163.7694, 197.2858, 175.8294},
	{233.105, 132.2032, 202.2302, 100.1675, 163.7694, 198.6258, 175.8294},
	{233.105, 166.8724, 234.6511, 100.1675, 163.7694, 198.6258, 206.9203},
	{228.305, 132.5732, 234.6511, 100.1675, 163.7694, 198.6258, 207.2511},
	{232.405, 164.9941, 234.6511, 100.1675, 163.7694, 199.9713, 207.2511},
	{233.405, 164.9941, 199.6511, 100.1675, 163.7694, 198.2858, 175.4602},
	{233.405, 131.0249, 199.6511, 100.1675, 165.1094, 199.9713, 210.4602},
	{233.405, 131.0249, 199.6511, 100.1675, 165.1094, 200.8258, 210.4602},
	{233.405, 131.0249, 199.6511, 100.1675, 131.9885, 200.8258, 210.4602},
	{233.405, 130.3249, 199.6511, 100.1675, 133.2885, 134.4357, 210.4602},
	{200.9841, 131.3249, 199.6511, 100.1675, 133.2885, 168.4049, 210.4602},
	{201.2841, 131.3249, 167.0274, 100.1675, 132.5885, 168.4049, 210.4602},
	{201.2841, 131.3249, 199.3111, 100.1675, 132.5885, 168.4049, 211.1602},
	{236.9141, 131.3249, 200.9966, 100.1675, 134.9285, 167.7749, 211.1602},
	{201.2594, 131.3249, 200.9966, 98.8375, 133.2985, 200.1958, 211.1602},
	{167.2902, 131.3249, 200.9966, 131.2584, 135.6285, 200.1958, 209.8302},
	{157.6902, 131.3249, 200.9966, 129.5729, 169.5977, 202.8813, 241.2511},
	{123.721, 131.3249, 202.3421, 129.5729, 169.5977, 200.8958, 241.2511},
	{128.521, 131.3249, 200.6966, 129.5729, 169.5977, 204.0813, 241.2511},
	{130.021, 131.3249, 167.1966, 129.5729, 169.5977, 204.0813, 241.2511},
	{134.821, 132.0249, 134.7757, 129.5729, 169.5977, 170.1121, 241.2511},
	{136.321, 133.5249, 135.0757, 129.5029, 169.5977, 170.1121, 241.2511},
	{137.021, 133.5249, 134.7757, 199.1721, 169.5977, 170.1121, 241.2511},
	{138.521, 101.104, 136.2757, 199.1721, 169.5977, 170.1121, 207.2819},
	{171.321, 101.104, 136.2757, 201.3721, 169.5977, 170.1121, 207.2819},
	{171.321, 99.774, 136.2757, 232.8013, 134.5977, 170.1121, 207.2819},
	{171.321, 99.774, 137.2812, 199.8176, 134.5977, 170.1121, 207.2819},
	{171.321, 132.1949, 138.9667, 234.8176, 134.5977, 204.4121, 207.2819},
	{171.321, 132.1949, 137.6212, 234.8176, 134.5977, 204.4121, 207.2819},
	{171.321, 132.1949, 138.6212, 234.8176, 134.5977, 204.4121, 207.2819},
	{171.321, 132.1949, 138.6212, 233.1321, 134.5977, 204.4121, 137.2819},
	{171.321, 132.1949, 138.6212, 236.6721, 169.8969, 204.4121, 137.9819},
	{167.851, 132.1949, 138.6212, 235.6721, 169.8969, 204.4121, 137.9819},
	{206.951, 167.8249, 104.652, 234.3321, 170.2277, 204.4121, 137.2819},
	{206.951, 167.8249, 104.652, 236.0176, 170.2277, 171.9912, 139.861},
	{206.251, 167.4941, 104.652, 235.6776, 170.2277, 138.022, 139.861},
	{207.251, 167.4941, 104.652, 204.9422, 136.2585, 138.022, 139.861},
	{202.451, 167.4941, 105.352, 204.9422, 136.2585, 138.022, 139.861},
	{241.551, 167.4941, 105.352, 202.7422, 136.2585, 138.022, 139.861},
	{206.551, 167.4941, 104.652, 203.7422, 168.6794, 136.692, 138.821},
	{206.551, 167.4941, 139.652, 203.7422, 168.6794, 172.322, 140.5065},
	{206.551, 165.8086, 139.652, 202.0567, 168.6794, 203.4129, 139.8765},
	{206.551, 200.1086, 139.652, 200.3712, 168.6794, 203.4129, 138.3765},
	{206.551, 200.1086, 139.652, 200.3712, 168.6794, 203.4129, 170.7974},
	{206.551, 200.1086, 139.652, 200.3712, 168.6794, 203.4129, 170.7974},
	{206.551, 164.4786, 139.652, 166.402, 168.6794, 170.992, 170.7974},
	{204.8655, 196.8995, 137.9665, 166.402, 168.3339, 235.8338, 169.4674},
	{204.8655, 196.8995, 136.9665, 131.402, 168.3339, 235.8338, 169.4674},
	{169.8655, 199.7778, 136.9665, 129.902, 168.3339, 235.8338, 169.4674},
	{169.8655, 199.7778, 136.9665, 129.902, 168.3339, 235.8338, 170.7974},
	{166.1055, 199.7778, 136.3365, 165.532, 168.3339, 200.8338, 204.7666},
	{169.8655, 200.4778, 168.7574, 130.532, 168.3339, 200.8338, 204.7666},
	{169.291, 234.447, 168.7574, 130.532, 168.3339, 199.8338, 204.7666},
	{169.291, 234.447, 168.7574, 130.532, 167.2784, 199.8338, 204.7666},
	{174.091, 234.447, 167.2574, 130.532, 166.6484, 199.8338, 204.7666},
	{208.0602, 234.447, 167.9574, 130.532, 199.0693, 200.1338, 239.7666},
	{208.0602, 200.4778, 169.4574, 130.532, 234.0693, 200.1338, 239.7666},
	{208.0602, 236.1078, 169.4574, 130.532, 201.6484, 197.4483, 204.7666},
	{206.5602, 234.4223, 169.4574, 130.532, 201.6484, 198.4483, 205.4666},
	{206.5602, 234.4223, 201.8783, 130.532, 166.6484, 198.4483, 240.1358},
	{171.5602, 233.4223, 201.8783, 130.532, 166.6484, 198.4483, 277.2658},
	{171.5602, 231.7368, 202.5783, 130.532, 166.6484, 198.4483, 244.8449},
	{171.5602, 231.7368, 202.5783, 130.532, 166.6484, 198.4483, 243.1594},
	{167.4602, 231.7368, 201.2483, 130.532, 166.6484, 198.4483, 243.1594},
	{167.4602, 231.7368, 233.6692, 130.532, 166.6484, 166.0274, 243.1594},
	{167.4602, 194.5159, 233.6692, 130.532, 166.6484, 166.0274, 243.1594},
	{132.4602, 194.5159, 198.6692, 130.532, 166.6484, 97.1065, 242.4594},
	{137.2602, 233.6159, 198.6692, 130.532, 166.6484, 97.1065, 242.4594},
	{171.2294, 233.6159, 166.2483, 129.032, 166.6484, 97.1065, 240.9594},
	{171.2294, 199.6467, 166.2483, 129.032, 166.6484, 97.1065, 240.9594},
	{171.2294, 199.6467, 166.2483, 129.032, 166.6484, 97.1065, 240.6194},
	{171.2294, 199.6467, 166.2483, 129.032, 164.9629, 97.1065, 207.1357},
	{164.7439, 199.6467, 166.2483, 129.032, 164.9629, 97.1065, 207.1357},
	{160.6439, 165.6775, 166.2483, 129.032, 164.9629, 96.1065, 207.1357},
	{160.6439, 165.6775, 166.2483, 129.032, 130.8565, 96.1065, 207.1357},
	{130.4347, 165.6775, 166.2483, 94.032, 130.8565, 131.4057, 207.1357},
	{132.1202, 165.6775, 200.5483, 94.032, 164.8257, 131.4057, 207.1357},
	{136.2202, 165.6775, 200.5483, 129.032, 166.5112, 132.0357, 207.1357},
	{171.2202, 163.992, 131.6274, 131.572, 166.5112, 132.0357, 242.4349},
	{166.4202, 163.992, 168.8274, 130.7175, 131.5112, 132.7357, 242.4349},
	{171.2202, 128.992, 168.8274, 132.403, 131.5112, 133.6057, 208.4657},
	{172.7202, 128.992, 167.3274, 132.403, 131.5112, 166.0266, 206.7802},
	{172.7202, 163.292, 137.9065, 132.403, 131.5112, 165.3966, 171.7802},
	{172.7202, 163.292, 137.9065, 132.403, 131.5112, 197.8175, 171.7802},
	{172.7202, 163.292, 137.9065, 168.733, 131.5112, 197.8175, 171.7802},
	{172.7202, 163.292, 137.9065, 202.7022, 131.5112, 197.8175, 171.7802},
	{171.7202, 161.6065, 137.9065, 202.7022, 131.5112, 197.8175, 136.7802},
	{171.7202, 161.6065, 137.9065, 202.7022, 131.5112, 197.8175, 136.1502},
	{171.7202, 161.6065, 137.9065, 202.7022, 129.8257, 233.1167, 167.0711},
	{167.6202, 161.6065, 137.9065, 204.3877, 129.8257, 233.1167, 167.0711},
	{167.6202, 161.6065, 137.9065, 205.2422, 129.8257, 233.1167, 167.0711},
	{172.4202, 161.6065, 137.9065, 205.2422, 129.8257, 233.1167, 167.0711},
	{172.4202, 164.1465, 137.9065, 205.2422, 129.8257, 231.6167, 167.0711},
	{172.4202, 164.1465, 137.2065, 205.2422, 129.8257, 231.6167, 167.0711},
	{172.4202, 129.1465, 138.2065, 205.9422, 129.8257, 231.6167, 167.0711},
	{174.9602, 129.1465, 137.5765, 239.9114, 129.8257, 231.6167, 169.6111},
	{174.9602, 128.1465, 138.9065, 239.9114, 129.8257, 197.6475, 168.4111},
	{174.9602, 129.1465, 172.8757, 239.9114, 130.5257, 197.6475, 165.8711},
	{174.9602, 131.1865, 172.8757, 239.9114, 166.5349, 197.6475, 167.5566},
	{174.9602, 129.8565, 172.8757, 239.2114, 166.5349, 197.6475, 133.5874},
	{174.9602, 163.6174, 172.8757, 205.2114, 166.5349, 165.2266, 133.5874},
	{139.9602, 163.6174, 172.8757, 203.8814, 166.5349, 164.2266, 133.5874},
	{135.8602, 163.6174, 208.1749, 203.8814, 165.1949, 162.5411, 133.5874},
	{135.8602, 161.9319, 208.1749, 203.8814, 166.8804, 162.5411, 133.5874},
	{140.6602, 160.9319, 208.1749, 203.5414, 166.8804, 130.1202, 131.0474},
	{142.1602, 160.9319, 173.1749, 203.5414, 202.1796, 131.1202, 132.7329},
	{142.1602, 125.9319, 173.1749, 203.5414, 200.6796, 131.1202, 100.942},
	{142.1602, 125.9319, 171.6749, 203.5414, 200.6796, 131.1202, 100.942},
	{142.1602, 125.9319, 206.6749, 201.9931, 165.3804, 130.1202, 135.6112},
	{142.1602, 127.2719, 206.6749, 166.9931, 197.8013, 131.1202, 135.6112},
	{142.1602, 127.2719, 209.2149, 166.9931, 197.8013, 166.4194, 138.1512},
	{142.1602, 125.5864, 209.2149, 166.9931, 196.1158, 166.4194, 138.1512},
	{142.1602, 126.9264, 209.2149, 166.9931, 196.1158, 132.1202, 138.1512},
	{103.391, 126.9264, 209.2149, 166.9931, 196.1158, 130.2719, 138.1512},
	{106.861, 126.9264, 240.1358, 200.9623, 196.1158, 131.7719, 138.1512},
	{139.2819, 125.2409, 240.1358, 200.9623, 196.1158, 131.7719, 138.1512},
	{139.2819, 125.2409, 240.1358, 201.2931, 197.8013, 131.7719, 138.1512},
	{134.4819, 125.2409, 241.6358, 201.2931, 197.8013, 133.1119, 169.2421},
	{138.2819, 157.6618, 207.6666, 201.2931, 196.1158, 131.7719, 136.8212},
	{172.2511, 157.6618, 207.6666, 167.3239, 196.1158, 133.4574, 168.6121},
	{172.2511, 157.6618, 207.6666, 167.3239, 194.6158, 133.4574, 168.6121},
	{172.2511, 125.2409, 207.6666, 167.3239, 194.6158, 132.8274, 166.6121},
	{172.2511, 125.2409, 207.6666, 167.3239, 160.6466, 132.8274, 166.6121},
	{172.2511, 125.2409, 207.6666, 167.3239, 127.0329, 132.8274, 166.6121},
	{172.2511, 126.9264, 173.6974, 169.0094, 159.4538, 132.8274, 199.033},
	{172.2511, 126.9264, 173.6974, 204.8094, 159.4538, 165.5483, 199.033},
	{172.2511, 158.0173, 173.6974, 170.5094, 159.4538, 164.8483, 197.533},
	{172.2511, 158.0173, 173.6974, 239.4786, 159.4538, 165.5483, 197.533},
	{172.2511, 126.9264, 173.6974, 207.0577, 127.0329, 167.0483, 196.833},
	{172.2511, 160.8956, 173.6974, 204.8577, 127.0329, 167.0483, 231.833},
	{172.2511, 160.8956, 173.6974, 205.8577, 127.0329, 167.0483, 197.8638},
	{172.2511, 160.8956, 138.6974, 204.8577, 127.0329, 133.2974, 197.8638},
	{172.2511, 160.8956, 139.3274, 204.8577, 127.0329, 165.7183, 197.8638},
	{172.2511, 160.8956, 106.9065, 203.3577, 127.0329, 164.2183, 197.8638},
	{171.2511, 160.8956, 106.9065, 203.3577, 127.0329, 162.5328, 197.8638},
	{138.8302, 160.5556, 137.9974, 203.3577, 162.6321, 162.5328, 197.8638},
	{172.7994, 197.5403, 105.5765, 203.3577, 162.6321, 162.5328, 197.8638},
	{172.7994, 130.4502, 172.9666, 203.3577, 161.2921, 162.5328, 165.4429},
	{172.7994, 200.4111, 172.9666, 203.3577, 162.9776, 198.1628, 165.4429},
	{172.7994, 197.8711, 172.9666, 203.3577, 162.9776, 198.1628, 165.4429},
	{172.7994, 199.5566, 172.9666, 168.3577, 162.9776, 196.8328, 165.4429},
	{168.6994, 199.5566, 171.2811, 168.3577, 163.6231, 229.2537, 166.7884},
	{168.6994, 199.5566, 171.2811, 168.3577, 163.6231, 229.2537, 165.4029},
	{167.1511, 199.5566, 171.2811, 168.3577, 165.3086, 232.4628, 133.6675},
	{167.1511, 199.5566, 171.2811, 168.3577, 165.3086, 234.1483, 170.1675},
	{167.1511, 234.2258, 171.2811, 167.3577, 131.2022, 234.1483, 170.1675},
	{205.9203, 234.2258, 170.2811, 167.3577, 132.8877, 234.1483, 170.1675},
	{205.9203, 200.2566, 170.2811, 167.3577, 132.8877, 234.1483, 170.1675},
	{205.9203, 236.7658, 168.7811, 133.3885, 132.8877, 234.1483, 170.1675},
	{200.3203, 235.5658, 168.7811, 133.3885, 132.8877, 234.1483, 169.1275},
	{205.1203, 235.5658, 168.7811, 133.3885, 132.8877, 232.6483, 170.813},
	{206.6203, 203.7966, 167.0956, 97.6885, 132.8877, 200.2274, 170.813},
	{204.0803, 203.7966, 167.0956, 98.0585, 166.8569, 232.6483, 170.813},
	{240.7658, 202.2966, 167.0956, 130.4794, 167.4869, 231.6083, 170.813},
	{240.7658, 203.7966, 167.0956, 130.4794, 236.1253, 233.2938, 170.813},
	{240.7658, 203.7966, 134.6747, 130.4794, 236.1253, 232.9483, 135.813},
	{239.2658, 238.7966, 134.6747, 130.4794, 202.1561, 232.9483, 135.813},
	{237.9358, 238.7966, 133.1747, 130.4794, 202.1561, 232.9483, 135.813},
	{270.3567, 238.7966, 133.1747, 130.4794, 202.1561, 232.9483, 135.813},
	{236.3875, 206.3757, 133.1747, 130.4794, 233.247, 200.5274, 171.1122},
	{236.3875, 206.3757, 99.2055, 128.7939, 233.247, 200.5274, 169.4267},
	{236.3875, 171.3757, 99.2055, 125.4229, 233.247, 165.5274, 169.4267},
	{202.9266, 171.3757, 99.2055, 125.4229, 233.247, 165.8274, 202.0967},
	{204.6121, 171.3757, 98.1655, 125.4229, 233.247, 233.2483, 202.0967},
	{202.9266, 171.3757, 99.851, 124.4229, 233.247, 233.2483, 167.0967},
	{204.6121, 169.8757, 99.851, 159.4229, 233.247, 232.9483, 202.0967},
	{204.6121, 169.8757, 99.851, 159.4229, 268.877, 234.4483, 203.4267},
	{170.6429, 169.8757, 99.851, 159.4229, 268.877, 234.4483, 237.3959},
	{170.6429, 135.9065, 99.851, 159.4229, 268.877, 198.4483, 202.3959},
	{170.6429, 135.9065, 99.851, 159.4229, 268.877, 198.4483, 202.3959},
	{170.6429, 135.9065, 98.851, 159.4229, 268.877, 166.0274, 202.3959},
	{170.6429, 135.9065, 98.851, 159.4229, 269.917, 165.0274, 202.3959},
	{165.8429, 135.9065, 98.851, 127.632, 270.217, 165.0274, 202.3959},
	{170.6429, 135.9065, 98.851, 127.632, 236.2478, 200.3266, 202.3959},
	{204.6121, 135.9065, 134.1502, 127.002, 235.2478, 200.3266, 202.3959},
	{204.6121, 135.9065, 132.8202, 159.4229, 235.2478, 200.3266, 202.3959},
	{204.6121, 135.9065, 165.2411, 159.4229, 167.3094, 166.3574, 202.3959},
	{204.6121, 135.9065, 165.2411, 159.4229, 167.3094, 200.6574, 202.3959},
	{204.6121, 135.9065, 165.2411, 159.4229, 167.3094, 200.6574, 202.3959},
	{167.3912, 100.9065, 165.2411, 159.4229, 167.3094, 200.6574, 202.3959},
	{135.8612, 100.9065, 165.2411, 159.4229, 167.3094, 200.6574, 237.6959},
	{166.7821, 100.9065, 165.2411, 159.4229, 167.3094, 168.2365, 202.3967},
	{166.7821, 100.9065, 163.7411, 159.4229, 167.3094, 168.2365, 203.7267},
	{165.7821, 100.9065, 163.7411, 159.4229, 167.3094, 168.2365, 272.9951},
	{165.7821, 169.8757, 163.7411, 195.0529, 167.3094, 168.2365, 273.0006},
	{159.9821, 169.8757, 163.7411, 195.0529, 134.8885, 167.2365, 273.3406},
	{159.9821, 169.8757, 164.3711, 194.3529, 134.8885, 168.922, 274.3406},
	{159.9821, 169.8757, 167.5566, 195.3529, 134.8885, 168.922, 274.3406},
	{162.0566, 135.9065, 167.5566, 195.3529, 134.8885, 167.2365, 240.3714},
	{163.7421, 169.8757, 165.0111, 195.3529, 99.8885, 133.922, 240.3714},
	{164.7421, 169.8757, 201.0111, 195.3529, 99.8885, 133.922, 242.0569},
	{161.2721, 168.8757, 236.0111, 195.3529, 99.8885, 133.922, 207.0569},
	{161.2721, 168.8757, 236.0111, 195.3529, 133.8577, 169.552, 205.3714},
	{200.0413, 168.8757, 236.0111, 160.3529, 133.8577, 169.552, 207.0569},
	{200.0413, 168.8757, 169.621, 128.632, 166.8269, 169.552, 207.7569},
	{200.0413, 168.8757, 169.621, 162.6012, 166.8269, 169.552, 207.5714},
	{200.0413, 167.8757, 169.621, 163.9412, 166.8269, 169.552, 207.5714},
	{200.7413, 198.9666, 169.621, 163.9412, 165.4969, 169.552, 207.5714},
	{168.2721, 197.9666, 170.961, 164.3112, 197.9178, 169.552, 207.5714},
	{132.3812, 162.0757, 166.161, 164.9412, 196.2878, 204.2212, 206.5714},
	{171.4812, 166.8757, 170.961, 199.9412, 228.7087, 239.5204, 206.5714},
	{171.4812, 200.8449, 171.461, 202.4812, 228.7087, 205.882, 206.5714},
	{171.4812, 200.8449, 206.461, 199.9412, 228.7087, 239.8512, 207.2714},
	{171.4812, 200.8449, 206.461, 202.4812, 228.7087, 204.8512, 206.2406},
	{171.4812, 200.8449, 206.461, 199.9412, 228.7087, 204.8512, 138.3022},
	{171.4812, 200.8449, 206.461, 201.6267, 227.7087, 204.8512, 138.3022},
	{171.4812, 200.8449, 206.461, 201.6267, 228.4087, 204.8512, 138.3022},
	{171.4812, 200.8449, 206.461, 166.6267, 231.2542, 204.5112, 138.3022},
	{171.4812, 200.8449, 205.8155, 166.6267, 230.6087, 206.1967, 138.3022},
	{169.9812, 131.8757, 203.2755, 166.6267, 231.1087, 206.1967, 138.3022},
	{169.9812, 131.8757, 203.961, 166.6267, 232.4542, 206.1967, 135.1167},
	{169.9812, 131.8757, 203.961, 166.6267, 233.3087, 206.1967, 135.1167},
	{169.9812, 131.8757, 203.961, 166.6267, 232.6632, 206.1967, 135.1167},
	{169.9812, 131.8757, 203.961, 165.2867, 233.1632, 206.8967, 135.1167},
	{169.9812, 131.8757, 203.961, 166.9722, 233.1632, 240.8659, 135.1167},
	{128.442, 131.8757, 203.261, 164.9467, 199.194, 204.3659, 135.1167},
	{171.642, 131.8757, 168.261, 132.663, 165.2248, 204.3659, 135.1167},
	{166.842, 131.8757, 132.631, 132.663, 131.1184, 204.3659, 135.1167},
	{171.642, 131.8757, 165.1819, 167.663, 131.1184, 204.3659, 135.1167},
	{173.142, 130.6757, 165.1819, 167.663, 131.1184, 204.3659, 135.1167},
	{173.142, 132.1757, 165.1819, 167.663, 134.6584, 204.3659, 135.1167},
	{173.142, 132.1757, 199.8511, 167.663, 102.2375, 204.3659, 135.1167},
	{173.142, 167.4749, 199.8511, 132.033, 136.5375, 204.3659, 135.1167},
	{173.142, 167.4749, 199.8511, 164.4539, 133.9975, 204.3659, 135.1167},
	{138.142, 133.5057, 199.8511, 129.4539, 135.683, 169.3659, 135.1167},
	{138.142, 133.5057, 200.5511, 129.4539, 169.6522, 135.3967, 135.1167},
	{138.142, 133.5057, 203.5511, 129.4539, 169.6522, 135.3967, 100.4475},
	{138.142, 133.5057, 166.7111, 129.4539, 169.6522, 135.3967, 101.1475},
	{138.142, 133.5057, 168.3966, 129.4539, 169.6522, 135.3967, 135.1167},
	{138.142, 133.5057, 168.3966, 129.4539, 169.6522, 135.3967, 135.1167},
	{138.142, 133.5057, 168.3966, 129.4539, 169.6522, 135.3967, 133.7867},
	{137.142, 133.5057, 167.0666, 129.4539, 169.6522, 135.3967, 166.2076},
	{137.142, 134.2057, 199.4875, 129.4539, 169.6522, 135.3967, 166.2076},
	{137.142, 134.2057, 198.7875, 129.4539, 169.6522, 135.3967, 164.7076},
	{137.142, 133.5057, 233.7875, 129.4539, 168.5967, 135.3967, 164.7076},
	{130.842, 168.5057, 268.7875, 127.7684, 202.5967, 135.3967, 164.7076},
	{130.842, 168.5057, 234.4875, 127.7684, 202.5967, 133.7112, 164.0076},
	{130.842, 168.5057, 268.4567, 127.7684, 200.9112, 99.742, 163.3776},
	{130.842, 167.5202, 271.335, 127.7684, 200.9112, 99.742, 195.7985},
	{134.312, 202.9894, 234.5358, 128.6229, 200.9112, 100.742, 195.7985},
	{166.7329, 202.9894, 266.9567, 96.202, 236.5412, 100.112, 195.7985},
	{161.9329, 202.9894, 266.9567, 96.202, 273.1859, 99.242, 195.7985},
	{126.9329, 202.9894, 266.9567, 128.6712, 271.5004, 134.242, 196.4985},
	{130.4029, 203.6894, 266.9567, 94.702, 273.1859, 134.242, 196.4985},
	{162.8238, 205.1894, 266.9567, 128.6712, 273.1859, 134.242, 196.4985},
	{154.2638, 205.1894, 266.9567, 161.0921, 204.9167, 134.242, 196.4985},
	{158.3638, 171.2202, 232.2875, 128.6712, 238.8859, 134.242, 196.1585},
	{165.6638, 170.5202, 267.9875, 161.0921, 238.8859, 134.242, 197.144},
	{165.6638, 171.2202, 269.4875, 161.0921, 238.8859, 134.242, 232.144},
	{161.5638, 205.1894, 270.4875, 161.0921, 238.8859, 134.242, 232.144},
	{166.3638, 205.1894, 269.4875, 163.6321, 238.8859, 134.242, 165.7539},
	{200.333, 205.1894, 270.4875, 198.6321, 238.8859, 168.542, 168.2939},
	{200.333, 205.1894, 238.0666, 165.3721, 238.8859, 167.542, 168.2939},
	{200.333, 205.1894, 238.0666, 200.8413, 238.8859, 167.542, 168.2939},
	{200.333, 205.1894, 238.0666, 200.8413, 238.8859, 133.242, 168.2939},
	{200.333, 205.1894, 238.0666, 200.8413, 238.8859, 165.7112, 170.8339},
	{200.333, 203.5039, 238.0666, 200.8413, 238.8859, 165.7112, 170.8339},
	{196.233, 203.5039, 203.0666, 200.8413, 238.8859, 165.7112, 138.413},
	{163.8121, 203.5039, 203.0666, 200.8413, 203.8859, 165.7112, 135.3975},
	{167.2821, 171.7439, 203.0666, 200.8413, 203.8859, 165.7112, 167.8184},
	{200.003, 172.0439, 203.0666, 200.8413, 203.8859, 167.0567, 167.8184},
	{200.003, 138.0747, 169.1457, 236.1405, 202.2004, 165.3712, 167.8184},
	{167.5821, 136.7347, 135.1765, 236.1405, 168.2312, 165.3712, 167.8184},
	{167.5821, 134.5347, 170.4757, 236.1405, 133.2312, 165.7112, 167.8184},
	{167.5821, 135.5347, 135.1765, 236.1405, 131.5457, 168.2112, 167.8184},
	{167.5821, 135.5347, 167.5974, 236.1405, 131.5457, 168.2112, 166.1329},
	{167.5821, 135.5347, 167.5974, 203.8568, 133.2312, 168.2112, 164.4329},
	{167.5821, 136.2347, 167.5974, 169.7504, 97.5765, 131.5257, 165.4329},
	{167.5821, 170.2039, 167.5974, 171.4359, 99.262, 131.5257, 165.4329},
	{167.5821, 168.8739, 167.8974, 171.4359, 100.2565, 131.5257, 165.4329},
	{167.5821, 135.5347, 167.5974, 171.4359, 100.2565, 131.5257, 165.4329},
	{167.5821, 170.5347, 168.0974, 170.4359, 100.2565, 131.5257, 165.4329},
	{167.5821, 170.5347, 167.0666, 170.4359, 100.2565, 130.8957, 165.4329},
	{132.9274, 170.5347, 167.3974, 170.4359, 101.5965, 197.2858, 128.9329},
	{132.9274, 170.5347, 167.6974, 170.4359, 102.7965, 195.6003, 128.9329},
	{132.9274, 169.5347, 168.3429, 170.4359, 102.7965, 195.6003, 128.9329},
	{132.9274, 169.5347, 167.0029, 170.4359, 103.311, 195.6003, 163.6021},
	{132.9274, 169.5347, 168.3429, 136.4667, 101.111, 162.9711, 128.9329},
	{132.9274, 168.0347, 168.3429, 136.4667, 102.111, 197.2711, 163.9329},
	{131.4274, 168.0347, 168.3429, 136.4667, 102.111, 197.2711, 131.512},
	{99.0065, 168.0347, 168.3429, 136.4667, 101.781, 197.2711, 163.9329},
	{99.0065, 203.0347, 168.3429, 136.4667, 168.1711, 197.2711, 163.9329},
	{99.0065, 203.0347, 168.3429, 102.4975, 168.1711, 197.2711, 163.9329},
	{99.0065, 203.0347, 168.3429, 102.4975, 168.1711, 198.7711, 163.9329},
	{99.0065, 203.0347, 166.6574, 102.4975, 168.1711, 197.2711, 164.2329},
	{97.321, 203.0347, 134.2365, 136.7975, 168.1711, 198.7711, 198.8229},
	{97.321, 203.0347, 134.2365, 101.1675, 168.1711, 198.7711, 201.5084},
	{97.321, 203.5347, 134.2365, 169.2184, 168.1711, 198.7711, 199.1684},
	{93.561, 203.5347, 134.2365, 203.1876, 168.1711, 198.7711, 201.8539},
	{93.561, 203.5347, 134.2365, 202.4876, 168.1711, 198.7711, 201.8539},
	{93.561, 202.3347, 134.2365, 202.4876, 168.1711, 198.7711, 200.8539},
	{91.8755, 202.3347, 134.2365, 237.4876, 168.1711, 199.4166, 200.8539},
	{91.8755, 167.3655, 134.2365, 237.4876, 168.1711, 198.7866, 234.8231},
	{126.8755, 167.3655, 134.2365, 237.4876, 168.1711, 231.2075, 234.8231},
	{160.2964, 132.3655, 134.2365, 237.4876, 168.1711, 197.1011, 234.8231},
	{164.3964, 133.7055, 134.2365, 237.4876, 168.1711, 198.7866, 234.8231},
	{165.3964, 133.7055, 166.6574, 237.4876, 203.1711, 164.8174, 234.8231},
	{165.3964, 132.7055, 131.6574, 237.4876, 168.5111, 164.8174, 235.4531},
	{165.3964, 132.7055, 131.6574, 237.4876, 203.5111, 164.8174, 235.4531},
	{165.3964, 135.2455, 131.6574, 237.4876, 173.2902, 165.8174, 234.8231},
	{165.3964, 135.2455, 131.6574, 237.4876, 173.2902, 167.2029, 267.244},
	{165.3964, 135.2455, 131.6574, 273.1331, 173.2902, 168.7029, 270.4531},
	{165.3964, 134.2455, 131.6574, 272.4876, 173.2902, 168.7029, 235.4531},
	{165.3964, 134.2455, 131.6574, 276.1876, 173.2902, 167.9029, 236.7931},
	{165.3964, 135.2455, 131.6574, 274.6876, 173.2902, 131.2029, 236.7931},
	{165.3964, 133.9055, 131.6574, 276.1876, 139.321, 165.2029, 236.7931},
	{161.6364, 135.591, 167.2874, 276.1876, 173.2902, 165.2029, 236.7931},
	{161.6364, 100.591, 202.2874, 243.7667, 173.2902, 165.2029, 235.1076},
	{161.6364, 100.591, 202.2874, 243.7667, 172.6602, 200.2029, 235.1076},
	{161.6364, 100.591, 202.2874, 243.7667, 205.0811, 165.2029, 235.1076},
	{161.6364, 100.591, 237.2874, 208.7667, 205.0811, 202.7429, 235.1076},
	{161.6364, 100.591, 237.2874, 174.7975, 205.0811, 202.7429, 200.1076},
	{200.0964, 94.461, 237.2874, 174.7975, 205.0811, 202.7429, 200.1076},
	{238.8656, 165.6511, 237.2874, 174.7975, 205.0811, 202.7429, 198.4221},
	{238.8656, 165.6511, 204.8665, 174.7975, 205.0811, 167.782, 200.1076},
	{238.8656, 130.9819, 204.8665, 174.7975, 205.0811, 169.4675, 200.9621},
	{238.8656, 165.9819, 204.8665, 139.7975, 205.0811, 204.7667, 166.9929},
	{238.8656, 199.9511, 204.8665, 138.7975, 203.7511, 205.0975, 166.9929},
	{238.8656, 199.9511, 204.8665, 137.112, 236.172, 205.0975, 166.9929},
	{238.8656, 199.9511, 204.8665, 137.112, 236.172, 205.0975, 166.9929},
	{203.8656, 199.9511, 204.8665, 137.112, 236.172, 203.412, 166.9929},
	{202.1801, 199.9511, 204.8665, 136.772, 202.512, 203.412, 134.572},
	{202.1801, 199.9511, 203.181, 138.4575, 202.512, 203.412, 134.572},
	{202.1801, 199.9511, 205.721, 138.4575, 202.512, 203.412, 134.572},
	{200.6801, 199.9511, 205.721, 138.4575, 238.142, 203.412, 98.072},
	{200.6801, 200.6511, 205.721, 138.4575, 238.142, 203.412, 98.072},
	{200.6801, 202.1511, 204.221, 138.4575, 238.142, 203.412, 99.7575},
	{200.6801, 202.1511, 204.221, 137.402, 238.142, 203.412, 99.7575},
	{197.5656, 202.1511, 204.221, 101.072, 204.1728, 167.782, 99.7575},
	{164.4447, 202.1511, 204.221, 137.0712, 171.7519, 200.2029, 99.7575},
	{165.4447, 202.1511, 204.221, 171.0404, 171.7519, 200.2029, 134.0575},
	{165.4447, 202.1511, 169.521, 171.0404, 171.7519, 199.2029, 134.0575},
	{201.3356, 202.1511, 169.521, 171.0404, 171.7519, 199.2029, 134.0575},
	{233.7565, 202.1511, 134.521, 169.3549, 171.7519, 197.5174, 98.4275},
	{233.7565, 169.3902, 134.521, 168.3549, 171.7519, 197.5174, 130.8484},
	{198.7565, 171.0757, 134.521, 169.0549, 171.7519, 198.8574, 165.8484},
	{198.7565, 171.0757, 134.521, 203.0241, 170.2519, 200.0574, 165.8484},
	{159.9873, 171.0757, 134.521, 203.0241, 170.2519, 165.0574, 165.8484},
	{159.9873, 170.0757, 99.521, 201.3386, 168.5664, 197.4783, 165.8484},
	{199.0873, 170.0757, 98.521, 201.3386, 136.1455, 197.4783, 165.8484},
	{199.0873, 136.1065, 98.521, 202.6786, 136.1455, 197.4783, 166.5484},
	{199.0873, 136.1065, 99.221, 202.6786, 136.1455, 162.4783, 200.5176},
	{199.0873, 136.8065, 133.1902, 201.3386, 136.1455, 196.7783, 200.5176},
	{199.0873, 169.4457, 168.1902, 203.0241, 136.1455, 231.7783, 200.5176},
	{199.0873, 166.8666, 168.1902, 203.0241, 136.1455, 231.7783, 200.5176},
	{199.0873, 166.8666, 168.1902, 203.0241, 136.1455, 231.7783, 200.5176},
	{199.0873, 166.8666, 168.1902, 203.0241, 134.8155, 231.7783, 200.5176},
	{199.0873, 166.5266, 168.1902, 203.0241, 167.2364, 231.7783, 200.5176},
	{199.0873, 168.2121, 168.1902, 203.0241, 167.2364, 199.3574, 200.5176},
	{199.0873, 168.9121, 168.1902, 203.0241, 163.1573, 199.3574, 200.5176},
	{199.0873, 203.8813, 167.3902, 203.0241, 163.1573, 199.3574, 200.5176},
	{199.0873, 202.8813, 168.8902, 169.0549, 162.1173, 199.3574, 200.5176},
	{199.0873, 203.8813, 168.8902, 169.0549, 163.8028, 199.3574, 200.5176},
	{134.2455, 203.8813, 168.8902, 135.0857, 163.8028, 200.3574, 200.5176},
	{134.2455, 203.8813, 168.8902, 137.6257, 162.3028, 200.3574, 168.0967},
	{134.2455, 203.8813, 168.8902, 137.6257, 162.3028, 200.3574, 166.4112},
	{134.2455, 203.8813, 168.8902, 137.6257, 162.3028, 200.3574, 166.4112},
	{134.2455, 203.8813, 168.8902, 137.9565, 162.3028, 167.9365, 166.4112},
	{134.2455, 203.8813, 167.2047, 139.642, 160.6173, 167.9365, 167.7512},
	{134.2455, 203.8813, 167.2047, 138.642, 160.6173, 167.9365, 167.7512},
	{129.2755, 203.8813, 167.2047, 138.642, 192.0382, 199.6574, 132.7512},
	{168.0447, 203.8813, 166.2047, 138.642, 190.5382, 200.6574, 132.7512},
	{168.0447, 171.4604, 166.2047, 104.342, 190.5382, 200.6574, 97.442},
	{168.0447, 169.9604, 132.2355, 139.6512, 190.5382, 200.3174, 99.1275},
	{133.0447, 169.9604, 132.2355, 139.6512, 158.1173, 202.0029, 131.5484},
	{133.0447, 169.9604, 132.2355, 139.6512, 158.1173, 167.0029, 131.5484},
	{133.0447, 134.4912, 132.2355, 139.6512, 158.1173, 167.0029, 128.8229},
	{133.0447, 169.1604, 133.2755, 139.6512, 126.3419, 131.3729, 130.5084},
	{133.0447, 135.1912, 98.921, 139.3112, 125.9964, 133.0429, 130.5084},
	{131.7147, 169.1604, 100.6065, 140.9967, 125.9964, 168.0429, 130.1684},
	{165.1356, 169.1604, 100.6065, 139.4967, 125.9964, 170.2429, 166.8539},
	{165.1356, 135.1912, 99.8065, 139.4967, 125.9964, 204.2121, 166.8539},
	{164.1356, 135.1912, 133.7757, 140.1967, 125.9964, 204.2121, 166.8539},
	{164.1356, 135.1912, 133.7757, 174.1659, 125.9964, 204.2121, 166.8539},
	{164.1356, 135.1912, 133.7757, 174.1659, 125.9964, 204.2121, 166.8539},
	{166.6756, 137.3212, 132.7757, 173.1659, 125.9964, 204.2121, 165.8539},
	{166.6756, 136.6912, 133.7757, 173.1659, 125.9964, 204.2121, 165.8539},
	{161.8756, 167.6121, 169.0749, 239.9351, 125.9964, 204.2121, 165.8539},
	{166.6756, 167.6121, 205.5749, 204.6359, 125.9964, 204.2121, 162.8539},
	{168.1756, 166.1121, 205.5749, 237.0568, 125.9964, 204.2121, 162.8539},
	{168.1756, 167.6121, 207.7749, 237.0568, 125.9964, 204.2121, 162.8539},
	{164.0756, 167.6121, 241.7441, 237.0568, 93.5755, 171.7912, 162.8539},
	{164.0756, 167.6121, 241.7441, 236.0568, 128.5364, 171.1612, 130.433},
	{126.0064, 167.6121, 239.5441, 236.0568, 126.6964, 203.5821, 130.093},
	{126.0064, 169.1121, 240.5441, 202.0876, 162.3511, 203.5821, 131.7785},
	{134.2764, 169.1121, 240.5441, 202.0876, 162.3511, 203.5821, 131.7785},
	{168.1973, 169.1121, 240.5441, 202.0876, 162.3511, 204.2821, 131.7785},
	{168.1973, 169.1121, 240.5441, 202.0876, 162.3511, 205.7821, 131.7785},
	{168.1973, 167.4266, 240.5441, 203.5876, 162.3511, 205.7821, 131.7785},
	{135.7764, 167.4266, 240.5441, 204.2876, 198.0511, 205.7821, 131.7785},
	{135.7764, 167.7266, 240.5441, 201.4576, 199.8511, 205.7821, 131.0785},
	{135.7764, 133.7574, 240.5441, 235.3785, 198.8511, 205.7821, 166.0785},
	{135.7764, 133.7574, 240.5441, 235.3785, 199.8511, 205.7821, 201.7085},
	{135.7764, 133.7574, 239.0441, 235.3785, 199.8511, 205.7821, 201.3777},
	{134.2764, 133.7574, 239.0441, 233.8785, 199.8511, 170.7821, 167.4085},
	{134.2764, 133.7574, 205.0749, 233.8785, 201.5366, 136.8129, 201.3777},
	{134.2764, 101.3365, 205.0749, 233.8785, 201.5366, 136.8129, 201.3777},
	{134.2764, 101.3365, 205.0749, 201.4093, 201.5366, 136.8129, 201.3777},
	{134.2764, 101.3365, 205.0749, 198.8693, 201.5366, 136.8129, 201.3777},
	{131.7764, 101.3365, 205.0749, 200.5548, 201.5366, 136.8129, 201.3777},
	{131.7764, 101.3365, 205.0749, 167.4339, 169.1157, 136.8129, 201.3777},
	{131.7764, 101.3365, 137.1365, 133.1339, 169.1157, 104.392, 201.3777},
	{131.7764, 137.8365, 137.1365, 167.1031, 169.1157, 104.392, 201.3777},
	{132.4764, 137.8365, 102.1365, 165.4176, 169.6157, 104.392, 201.3777},
	{130.5547, 136.8365, 134.751, 165.4176, 169.6157, 104.392, 201.3777},
	{169.6547, 136.8365, 134.751, 165.4176, 168.1157, 104.392, 201.3777},
	{169.6547, 138.1765, 134.751, 165.4176, 200.5366, 104.392, 201.3777},
	{169.6547, 136.8365, 134.421, 165.4176, 200.5366, 101.392, 201.3777},
	{169.6547, 138.522, 166.8419, 132.9967, 166.5674, 133.8129, 202.8777},
	{169.6547, 138.522, 166.8419, 132.9967, 166.5674, 136.6912, 203.0632},
	{164.8547, 138.522, 166.8419, 132.9967, 166.5674, 136.9912, 204.8632},
	{164.8547, 138.522, 166.8419, 132.9967, 166.5674, 135.3057, 204.8632},
	{164.8547, 138.522, 166.8419, 132.9967, 166.5674, 135.3057, 204.8632},
	{169.6547, 172.4912, 166.8419, 132.9967, 131.5674, 135.0057, 203.1777},
	{203.6239, 172.4912, 166.8419, 133.6967, 167.5666, 136.5057, 202.5477},
	{203.6239, 208.1212, 166.8419, 135.1967, 169.0666, 136.5057, 203.8777},
	{200.1539, 208.1212, 167.8419, 135.1967, 169.0666, 134.8202, 237.8469},
	{238.9231, 206.4357, 166.5019, 136.6967, 169.0666, 134.8202, 167.8469},
	{238.9231, 206.4357, 168.1874, 136.6967, 169.0666, 134.8202, 168.8777},
	{238.9231, 206.4357, 167.1874, 136.6967, 169.0666, 169.1202, 168.8777},
	{238.9231, 206.4357, 167.1874, 136.6967, 169.0666, 169.1202, 168.8777},
	{238.9231, 206.4357, 167.1874, 172.3267, 204.3658, 169.1202, 168.8777},
	{238.9231, 206.4357, 167.1874, 172.3267, 204.3658, 169.1202, 169.7322},
	{238.9231, 208.9757, 167.1874, 172.3267, 204.3658, 169.1202, 169.7322},
	{238.9231, 208.9757, 201.1566, 138.3575, 204.3658, 169.1202, 172.2722},
	{204.9539, 173.9757, 201.1566, 136.8575, 204.3658, 169.1202, 169.7322},
	{204.9539, 173.9757, 201.1566, 171.1575, 171.9449, 168.1202, 171.4177},
	{203.9539, 173.9757, 168.7357, 171.1575, 171.9449, 168.1202, 206.7169},
	{164.8539, 173.9757, 167.7357, 171.1575, 171.9449, 168.1202, 206.7169},
	{164.8539, 173.9757, 167.7357, 171.1575, 171.9449, 168.1202, 206.7169},
	{164.8539, 172.4757, 166.4057, 136.8575, 171.9449, 134.151, 206.7169},
	{164.8539, 172.4757, 198.8266, 170.8267, 171.9449, 135.491, 206.7169},
	{164.8539, 172.4757, 198.8266, 170.8267, 170.4449, 135.491, 206.7169},
	{164.8539, 173.4757, 198.8266, 206.1259, 170.4449, 135.491, 206.7169},
	{161.3839, 173.4757, 198.8266, 170.8267, 169.1149, 135.491, 206.7169},
	{127.4147, 139.5065, 198.8266, 203.2476, 169.7449, 135.491, 206.7169},
	{130.8847, 139.5065, 198.8266, 202.6176, 204.7449, 135.491, 205.3869},
	{163.3056, 139.5065, 198.8266, 202.6176, 171.4757, 135.491, 203.8386},
	{202.0748, 139.5065, 163.8266, 236.3785, 205.4449, 135.491, 203.8386},
	{202.0748, 139.5065, 163.8266, 236.3785, 205.4449, 135.491, 238.1386},
	{202.0748, 138.1765, 163.8266, 236.3785, 205.4449, 136.3455, 238.1386},
	{168.1056, 170.5974, 163.8266, 236.3785, 237.8658, 170.6455, 238.1386},
	{168.1056, 135.5974, 165.3266, 236.3785, 237.8658, 238.0664, 238.1386},
	{168.1056, 168.0183, 167.5266, 236.3785, 241.0749, 237.7356, 238.1386},
	{168.1056, 168.0183, 165.3266, 202.8785, 241.0749, 270.1565, 237.1386},
	{168.1056, 168.0183, 166.3266, 202.8785, 207.1057, 267.6165, 237.1386},
	{168.1056, 167.0183, 166.3266, 201.3785, 207.1057, 234.6328, 202.1386},
	{167.4056, 167.0183, 132.3574, 201.3785, 207.1057, 269.6328, 202.1386},
	{168.4056, 165.9783, 132.3574, 201.3785, 207.1057, 269.6328, 202.1386},
	{168.4056, 167.6638, 133.3574, 201.3785, 207.1057, 269.6328, 202.1386},
	{163.6056, 167.6638, 133.3574, 201.3785, 207.1057, 270.6328, 202.1386},
	{167.3656, 167.6638, 136.2357, 199.693, 207.1057, 272.6183, 202.1386},
	{169.0511, 167.6638, 136.2357, 167.2721, 207.1057, 272.3183, 202.1386},
	{169.0511, 167.6638, 136.2357, 133.3029, 207.1057, 273.8183, 202.1386},
	{164.9511, 167.6638, 136.9357, 133.9629, 207.1057, 273.8183, 168.1694},
	{164.9511, 167.6638, 170.9049, 135.6484, 207.1057, 273.8183, 135.7485},
	{169.0511, 167.6638, 170.9049, 103.2275, 207.1057, 273.8183, 135.7485},
	{137.6302, 167.6638, 169.4049, 103.2275, 206.1057, 273.8183, 135.7485},
	{137.6302, 135.2429, 171.9449, 103.2275, 206.1057, 273.8183, 134.2485},
	{137.6302, 133.7429, 170.4449, 103.2275, 206.1057, 273.8183, 134.2485},
	{137.6302, 133.7429, 170.4449, 103.2275, 206.1057, 273.8183, 134.2485},
	{103.661, 133.7429, 170.4449, 103.2275, 137.1365, 272.8183, 134.2485},
	{102.161, 99.6365, 170.7449, 103.2275, 137.1365, 238.8974, 134.2485},
	{102.161, 97.951, 170.7449, 101.8975, 137.1365, 206.4765, 97.563},
	{95.6755, 97.951, 170.7449, 134.3184, 137.1365, 206.4765, 98.903},
	{95.6755, 133.581, 170.7449, 134.3184, 137.4365, 206.4765, 98.903},
	{94.6755, 133.581, 170.7449, 134.3184, 135.7365, 171.4765, 102.643},
	{133.7755, 133.581, 170.7449, 134.3184, 170.7365, 171.4765, 101.443},
	{133.7755, 133.581, 170.7449, 134.3184, 170.4365, 136.4765, 101.443},
	{133.7755, 134.911, 169.7449, 134.3184, 136.9365, 136.4765, 101.443},
	{133.7755, 134.911, 169.7449, 134.3184, 136.9365, 136.4765, 100.113},
	{133.7755, 133.871, 205.0441, 134.3184, 136.9365, 136.4765, 100.113},
	{133.7755, 169.8565, 205.0441, 134.3184, 136.9365, 168.8974, 100.113},
	{159.1847, 169.8565, 205.0441, 132.6329, 136.9365, 168.8974, 100.113},
	{163.9847, 169.8565, 205.0441, 132.6329, 136.9365, 168.8974, 100.113},
	{203.0539, 169.8565, 171.0749, 132.6329, 135.251, 134.5974, 132.5339},
	{203.0539, 169.8565, 137.1057, 132.6329, 135.251, 133.8974, 132.5339},
	{203.0539, 168.8565, 137.1057, 132.6329, 134.251, 168.8974, 132.5339},
	{203.0539, 168.8565, 137.1057, 132.6329, 134.251, 168.8974, 129.8484},
	{201.0539, 168.8565, 169.9057, 132.6329, 135.751, 168.8974, 129.8484},
	{196.2539, 168.8565, 169.2057, 130.9474, 135.751, 168.8974, 129.8484},
	{200.3539, 168.8565, 204.2057, 130.9474, 135.751, 168.8974, 129.8484},
	{235.3539, 167.5165, 204.2057, 98.5265, 134.751, 168.8974, 129.8484},
	{235.3539, 169.202, 204.2057, 96.841, 134.751, 168.8974, 129.2184},
	{235.3539, 169.202, 204.2057, 96.841, 134.751, 168.8974, 162.3393},
	{235.3539, 169.202, 202.5202, 96.841, 134.751, 166.2119, 196.3085},
	{236.0539, 203.502, 202.5202, 96.841, 134.751, 166.2119, 196.3085},
	{237.5539, 203.502, 202.5202, 96.841, 134.751, 166.2119, 197.994},
	{237.5539, 167.872, 202.5202, 97.541, 134.751, 166.2119, 196.3085},
	{237.5539, 165.2929, 202.5202, 133.1957, 134.121, 166.2119, 194.623},
	{237.5539, 165.2929, 201.4802, 133.1957, 134.121, 166.2119, 196.3085},
	{237.5539, 165.2929, 203.1657, 133.1957, 134.121, 166.2119, 197.3085},
	{202.5539, 165.2929, 203.1657, 133.1957, 99.121, 166.2119, 197.3085},
	{202.5539, 199.9621, 203.1657, 133.1957, 99.121, 133.791, 197.3085},
	{168.5847, 199.9621, 169.1965, 130.6557, 99.121, 134.131, 197.3085},
	{168.5847, 199.9621, 169.1965, 132.3412, 97.791, 135.291, 197.3085},
	{134.6155, 165.9929, 169.1965, 132.3412, 97.1455, 134.7765, 164.8876},
	{133.6155, 165.9929, 169.1965, 167.9712, 98.4055, 136.4065, 164.8876},
	{133.6155, 130.9929, 169.1965, 167.9712, 167.3655, 136.4065, 164.8876},
	{133.6155, 130.2929, 169.1965, 169.3112, 169.051, 171.0757, 162.5476},
	{133.6155, 165.2929, 169.8965, 169.3112, 171.951, 171.0757, 162.5476},
	{133.6155, 166.8629, 203.8657, 169.3112, 171.951, 169.5757, 162.5476},
	{133.6155, 195.5838, 202.1802, 170.6512, 172.121, 204.5757, 162.5476},
	{133.6155, 196.5838, 202.1802, 170.6512, 204.5419, 135.2757, 160.8621},
	{132.6155, 196.5838, 131.4802, 204.2721, 204.5419, 169.2449, 196.1613},
	{97.6155, 196.5838, 131.4802, 204.2721, 204.5419, 169.2449, 196.4613},
	{97.6155, 196.5838, 130.4802, 204.2721, 204.5419, 169.2449, 196.4613},
	{96.1155, 197.9238, 131.1802, 204.2721, 204.5419, 169.2449, 196.4613},
	{96.1155, 165.5029, 166.1494, 204.2721, 204.5419, 169.2449, 162.4921},
	{96.1155, 165.5029, 199.1186, 204.2721, 206.2274, 169.2449, 162.8321},
	{96.1155, 165.5029, 200.1186, 204.2721, 241.2274, 169.2449, 162.4921},
	{130.4155, 165.5029, 200.1186, 170.3029, 241.2274, 169.2449, 164.1776},
	{130.4155, 165.5029, 200.1186, 170.3029, 240.2274, 171.4449, 164.1776},
	{130.4155, 166.8429, 200.1186, 204.2721, 240.2274, 169.9449, 164.1776},
	{130.4155, 166.8429, 200.1186, 238.2413, 240.2274, 171.4449, 164.1776},
	{126.9455, 167.5429, 200.1186, 238.2413, 240.2274, 171.4449, 163.5476},
	{165.7147, 201.5121, 198.6186, 238.2413, 240.2274, 171.4449, 195.9685},
	{200.0147, 201.5121, 198.6186, 238.2413, 240.2274, 171.4449, 195.9685},
	{200.0147, 201.5121, 198.6186, 238.2413, 240.2274, 171.4449, 197.3085},
	{195.9147, 201.5121, 198.6186, 238.2413, 238.5419, 171.4449, 197.3085},
	{195.9147, 201.5121, 198.6186, 238.2413, 238.5419, 137.4757, 197.3085},
	{195.9147, 201.5121, 164.6494, 236.5558, 203.5419, 136.8457, 197.3085},
	{199.6747, 199.8266, 164.6494, 201.5558, 171.121, 169.2666, 164.8876},
	{202.8602, 130.2757, 163.3194, 204.4341, 136.121, 169.2666, 164.8876},
	{202.8602, 162.6966, 163.3194, 169.1349, 136.121, 169.2666, 164.8876},
	{202.8602, 162.6966, 163.3194, 202.8958, 136.121, 135.2974, 164.8876},
	{202.8602, 162.6966, 164.6594, 204.0958, 171.751, 135.2974, 130.9184},
	{201.3602, 162.6966, 165.2894, 204.0958, 171.751, 135.2974, 130.9184},
	{201.3602, 162.6966, 200.2894, 204.0958, 171.751, 135.2974, 130.9184},
	{197.2602, 162.6966, 166.3202, 204.0958, 171.751, 135.2974, 130.9184},
	{201.6602, 162.6966, 166.3202, 204.7413, 171.751, 134.6674, 130.9184},
	{237.3602, 161.6966, 166.3202, 203.2413, 171.751, 167.0883, 129.2329},
	{238.8602, 161.6966, 166.3202, 201.8958, 171.751, 166.7883, 129.2329},
	{237.3602, 162.0366, 166.3202, 202.8958, 171.751, 168.2883, 129.2329},
	{237.3602, 162.0366, 132.351, 202.8958, 172.751, 168.2883, 129.2329},
	{202.3602, 162.0366, 132.351, 168.9266, 172.411, 166.7883, 129.2329},
	{202.3602, 162.0366, 132.351, 134.9574, 172.411, 166.7883, 96.812},
	{164.291, 157.9366, 132.351, 134.9574, 172.5965, 166.7883, 96.812},
	{168.391, 128.7129, 130.6655, 134.9574, 137.5965, 166.7883, 96.812},
	{165.291, 128.0274, 161.7564, 134.9574, 137.5965, 166.7883, 96.812},
	{129.591, 129.7129, 161.7564, 200.3475, 137.5965, 134.3674, 130.7812},
	{134.351, 129.7129, 161.7564, 200.3475, 137.5965, 134.3674, 130.7812},
	{170.0057, 129.7129, 161.7564, 200.3475, 136.0965, 134.3674, 131.7812},
	{170.0057, 97.292, 129.3355, 200.3475, 136.0965, 134.3674, 131.7812},
	{170.0057, 97.292, 129.3355, 200.3475, 136.0965, 132.1674, 131.7812},
	{170.0057, 97.292, 129.3355, 198.8475, 136.0965, 132.1674, 131.7812},
	{170.0057, 97.292, 161.7564, 166.4266, 134.5965, 167.1674, 130.4512},
	{170.0057, 95.792, 162.4564, 166.4266, 134.5965, 168.6674, 162.8721},
	{165.9057, 95.792, 163.9564, 167.9266, 134.5965, 168.6674, 162.8721},
	{165.9057, 95.792, 163.9564, 168.9266, 134.5965, 201.0883, 161.3721},
	{165.9057, 97.292, 164.2964, 168.9266, 135.5965, 168.6674, 161.3721},
	{165.9057, 97.292, 165.2964, 169.9666, 101.2965, 168.6674, 163.0576},
	{165.9057, 97.292, 166.6364, 167.4266, 101.5965, 167.6674, 163.0576},
	{170.7057, 97.292, 130.2964, 170.6121, 100.8965, 167.6674, 163.9121},
	{204.6749, 97.292, 131.9819, 170.6121, 135.8965, 167.6674, 163.9121},
	{169.6749, 96.092, 131.9819, 170.6121, 135.8965, 166.9674, 165.4121},
	{169.6749, 96.092, 131.9819, 170.6121, 135.8965, 168.6674, 163.9121},
	{169.6749, 131.722, 131.9819, 169.1121, 135.8965, 202.3366, 165.4121},
	{169.6749, 131.722, 131.2819, 169.1121, 135.8965, 203.8366, 201.0421},
	{169.6749, 131.722, 167.7819, 136.6912, 135.8965, 203.8366, 201.0421},
	{169.6749, 132.3675, 167.7819, 136.6912, 135.8965, 202.1511, 201.0421},
	{169.6749, 132.3675, 168.4819, 136.6912, 135.8965, 202.1511, 201.0421},
	{169.6749, 164.1584, 169.9819, 102.722, 135.8965, 202.1511, 202.3876},
	{135.0057, 196.5793, 169.9819, 102.722, 135.8965, 203.4911, 201.7421},
	{135.6657, 194.2083, 169.9819, 136.6912, 135.8965, 203.4911, 136.852},
	{135.6657, 194.3938, 137.561, 136.6912, 135.8965, 203.4911, 136.852},
	{135.6657, 194.3938, 137.561, 136.6912, 134.8965, 203.4911, 170.982},
	{135.6657, 194.3938, 137.561, 136.6912, 134.8965, 203.4911, 170.982},
	{135.6657, 194.3938, 137.561, 136.6912, 134.8965, 202.4511, 170.982},
	{135.6657, 194.3938, 136.561, 136.6912, 134.8965, 171.7157, 169.652},
	{135.6657, 194.3938, 136.561, 136.6912, 137.4365, 171.7157, 169.652},
	{135.6657, 194.3938, 136.561, 136.6912, 134.8965, 171.7157, 202.0729},
	{135.6657, 195.0238, 136.561, 136.6912, 136.582, 171.7157, 202.0729},
	{135.6657, 195.0238, 136.561, 136.6912, 136.582, 136.7157, 202.0729},
	{135.6657, 230.0238, 136.561, 136.6912, 136.582, 135.2157, 202.0729},
	{101.6965, 229.3938, 136.561, 136.6912, 135.882, 135.2157, 202.0729},
	{101.6965, 260.8147, 136.561, 136.6912, 136.882, 133.5302, 202.0729},
	{101.6965, 260.8147, 136.561, 136.6912, 136.882, 133.5302, 202.0729},
	{101.6965, 260.8147, 171.561, 136.6912, 136.882, 98.861, 202.0729},
	{101.6965, 260.8147, 171.561, 136.9912, 101.882, 99.491, 202.0729},
	{100.6965, 225.8147, 135.931, 135.9912, 101.882, 98.861, 202.7029},
	{100.6965, 193.3938, 168.3519, 133.6757, 101.882, 130.6519, 202.0729},
	{100.6965, 160.9729, 133.3519, 166.0966, 100.882, 163.0728, 234.4938},
	{100.6965, 193.3938, 165.7728, 166.0966, 100.882, 163.0728, 234.4938},
	{100.6965, 194.3938, 169.3511, 166.0966, 100.252, 163.0728, 199.4938},
	{100.6965, 194.3938, 202.3203, 166.7266, 134.552, 163.0728, 200.5338},
	{100.6965, 193.0538, 202.3203, 166.0966, 136.882, 163.0728, 200.5338},
	{100.6965, 194.7393, 201.6203, 198.5175, 170.8512, 163.7028, 200.5338},
	{100.6965, 195.5938, 236.6203, 198.5175, 170.8512, 198.7028, 200.8338},
	{100.6965, 195.5938, 236.6203, 164.5483, 170.8512, 197.2028, 200.8338},
	{100.6965, 195.5938, 235.1203, 164.5483, 170.8512, 197.8328, 200.8338},
	{100.6965, 195.5938, 234.1203, 164.5483, 170.8512, 232.8328, 168.4129},
	{96.5965, 195.5938, 234.1203, 164.5483, 170.8512, 232.1328, 132.7829},
	{134.0357, 195.5938, 234.1203, 164.5483, 170.8512, 232.8328, 165.2038},
	{166.4566, 195.5938, 234.1203, 164.5483, 169.3512, 234.3328, 165.2038},
	{166.4566, 197.0938, 234.1203, 164.5483, 169.3512, 235.6783, 165.2038},
	{166.4566, 201.0129, 234.1203, 199.8883, 169.3512, 235.6783, 165.2038},
	{166.4566, 166.0129, 234.1203, 199.8883, 204.3512, 235.6783, 165.2038},
	{166.4566, 166.0129, 234.1203, 199.8883, 204.0112, 235.6783, 165.2038},
	{166.4566, 166.0129, 234.1203, 199.8883, 205.6967, 235.6783, 163.7038},
	{166.4566, 166.0129, 201.6994, 200.8883, 205.6967, 235.0328, 163.7038},
	{166.4566, 133.592, 201.6994, 203.7666, 205.6967, 236.5328, 163.7038},
	{200.4258, 133.592, 201.6994, 203.7666, 205.6967, 171.691, 131.2829},
	{200.4258, 131.9065, 201.6994, 203.7666, 205.6967, 171.691, 131.2829},
	{200.4258, 131.9065, 201.6994, 203.7666, 205.6967, 171.691, 165.2274},
	{200.4258, 131.9065, 167.7302, 203.7666, 205.6967, 171.691, 165.2274},
	{200.4258, 133.2465, 166.0447, 239.0658, 205.6967, 172.031, 164.8966},
	{201.7658, 133.2465, 132.0755, 171.3457, 173.2275, 172.031, 164.8966},
	{201.7658, 133.2465, 132.0755, 203.7666, 173.2275, 174.231, 164.8966},
	{201.7658, 133.2465, 132.0755, 203.7666, 173.2275, 174.231, 163.8966},
	{201.7658, 131.9065, 132.0755, 203.7666, 171.0975, 173.531, 163.8966},
	{169.3449, 135.092, 132.0755, 204.2666, 203.5184, 174.531, 129.7902},
	{165.2449, 167.5129, 132.0755, 200.0411, 203.5184, 174.531, 165.4202},
	{165.2449, 164.0429, 132.0755, 201.7266, 168.5184, 174.531, 165.4202},
	{165.2449, 203.1429, 97.0755, 202.3721, 168.5184, 174.531, 165.7202},
	{165.2449, 203.1429, 97.0755, 201.0266, 168.5184, 139.531, 165.7202},
	{168.7149, 235.5638, 97.0755, 202.0266, 167.8884, 104.531, 165.7202},
	{201.1358, 235.5638, 97.0755, 202.0266, 200.3093, 104.531, 164.7202},
	{167.1666, 235.5638, 97.0755, 201.6866, 200.3093, 104.531, 165.7202},
	{167.1666, 235.5638, 97.0755, 203.3721, 200.3093, 104.3455, 165.7202},
	{167.1666, 235.5638, 96.7355, 203.3721, 200.3093, 104.3455, 165.7202},
	{163.0666, 235.5638, 98.421, 201.6866, 200.3093, 104.3455, 165.7202},
	{163.0666, 235.5638, 129.5119, 166.6866, 200.3093, 104.3455, 165.7202},
	{167.8666, 235.5638, 98.421, 166.6866, 165.3093, 104.3455, 164.0347},
	{163.0666, 200.5638, 132.3902, 165.6866, 165.3093, 104.3455, 164.0347},
	{163.0666, 200.5638, 133.3902, 165.6866, 167.5093, 104.3455, 164.0347},
	{163.0666, 200.5638, 133.3902, 133.2657, 168.2093, 104.3455, 164.0347},
	{167.8666, 200.5638, 133.3902, 133.2657, 166.5238, 104.3455, 164.0347},
	{201.8358, 200.5638, 132.3902, 133.2657, 165.8238, 136.7664, 196.4556},
	{201.8358, 200.5638, 133.3902, 99.2965, 200.8238, 136.7664, 164.0347},
	{201.8358, 200.5638, 133.3902, 132.5657, 197.1238, 135.7664, 162.4864},
	{200.3358, 200.5638, 133.6902, 167.5657, 166.0029, 135.7664, 162.4864},
	{200.3358, 168.1429, 133.6902, 167.5657, 166.0029, 135.7664, 160.8164},
	{200.3358, 168.1429, 132.3902, 167.5657, 164.3174, 135.7664, 162.5019},
	{200.3358, 168.1429, 133.8902, 167.5657, 164.3174, 135.7664, 162.5019},
	{200.3358, 135.722, 133.8902, 167.5657, 131.8965, 135.7664, 163.1319},
	{200.3358, 135.722, 133.8902, 167.5657, 131.8965, 135.7664, 198.1319},
	{167.9149, 135.722, 133.8902, 167.5657, 131.8965, 135.7664, 198.1319},
	{167.9149, 100.722, 133.8902, 167.5657, 131.8965, 134.2664, 163.1319},
	{167.9149, 100.722, 133.8902, 167.5657, 131.8965, 169.2664, 163.1319},
	{166.2294, 100.722, 133.8902, 167.5657, 131.8965, 133.0064, 162.5019},
	{165.2294, 100.722, 134.5202, 167.5657, 131.8965, 165.4273, 194.9228},
	{165.2294, 100.722, 133.8902, 167.9057, 164.3174, 165.4273, 193.9228},
	{165.2294, 99.722, 166.3111, 168.9057, 164.3174, 165.4273, 193.9228},
	{165.2294, 99.722, 165.3111, 168.9057, 164.3174, 165.4273, 193.9228},
	{165.2294, 135.352, 165.3111, 168.9057, 164.3174, 165.4273, 193.9228},
	{165.2294, 136.122, 131.3419, 168.9057, 197.0866, 134.3364, 193.9228},
	{123.6902, 171.5912, 131.3419, 168.9057, 197.0866, 168.3056, 161.5019},
	{162.7902, 172.2212, 131.3419, 170.2457, 198.4266, 168.3056, 161.5019},
	{133.621, 207.2212, 131.3419, 168.7457, 198.4266, 168.3056, 161.5019},
	{135.121, 207.9212, 130.0119, 168.7457, 198.4266, 168.3056, 161.5019},
	{135.121, 207.2212, 162.4328, 168.7457, 164.4574, 203.9356, 161.5019},
	{135.121, 242.2212, 162.4328, 168.7457, 198.7721, 203.9356, 161.5019},
	{134.121, 242.2212, 163.7728, 134.7765, 200.4576, 203.9356, 163.5419},
	{134.121, 242.2212, 163.7728, 134.7765, 232.8785, 203.9356, 166.2419},
	{134.121, 242.2212, 162.7728, 134.7765, 231.193, 203.9356, 168.7819},
	{133.121, 242.2212, 163.9728, 98.2765, 196.193, 203.9356, 168.7819},
	{133.121, 242.2212, 198.642, 98.2765, 196.193, 238.9356, 168.7819},
	{131.621, 242.2212, 198.642, 133.2765, 196.193, 238.9356, 168.7819},
	{131.621, 242.2212, 163.9728, 134.6065, 196.193, 205.5147, 168.7819},
	{130.121, 242.2212, 198.9728, 134.6065, 196.193, 241.1447, 168.7819},
	{130.121, 242.2212, 198.9728, 168.9065, 196.193, 242.4847, 171.6602},
	{130.121, 242.2212, 198.9728, 168.9065, 196.193, 242.4847, 171.6602},
	{130.121, 240.5357, 167.2519, 168.9065, 163.7721, 242.4847, 173.3457},
	{122.551, 277.5204, 170.0974, 204.9057, 163.7721, 242.4847, 138.3457},
	{156.851, 277.5204, 170.0974, 238.8749, 163.7721, 242.4847, 138.3457},
	{160.321, 277.5204, 170.6119, 238.8749, 163.7721, 240.9847, 138.3457},
	{192.7419, 277.5204, 169.7574, 237.1894, 163.7721, 240.9847, 173.9757},
	{196.5019, 242.5204, 169.7574, 237.1894, 163.7721, 207.0155, 173.6449},
	{198.1874, 242.5204, 169.7574, 237.1894, 163.7721, 207.0155, 173.6449},
	{198.1874, 208.5512, 137.3365, 237.1894, 163.7721, 207.0155, 173.6449},
	{232.1566, 208.5512, 137.3365, 237.1894, 163.7721, 207.0155, 173.6449},
	{232.1566, 208.5512, 137.3365, 237.1894, 131.3512, 207.0155, 209.2749},
	{187.5566, 173.5512, 137.3365, 237.1894, 130.7212, 206.6755, 209.2749},
	{191.3166, 173.5512, 137.3365, 237.1894, 163.1421, 206.6755, 209.2749},
	{193.0021, 138.5512, 137.3365, 237.1894, 129.1729, 206.6755, 209.2749},
	{192.0876, 138.5512, 137.3365, 237.1894, 129.1729, 206.6755, 242.9041},
	{196.8876, 138.5512, 137.3365, 237.1894, 129.1729, 172.0155, 242.9041},
	{230.8568, 138.5512, 137.3365, 237.1894, 129.1729, 173.0155, 242.9041},
	{229.1713, 138.5512, 137.3365, 237.1894, 129.1729, 174.0155, 242.9041},
	{229.1713, 138.5512, 137.3365, 239.3894, 129.1729, 138.7155, 242.9041},
	{232.9313, 138.5512, 172.3365, 204.3894, 162.9338, 140.2155, 242.9041},
	{234.6168, 138.5512, 207.2665, 200.3494, 162.9338, 140.2155, 241.4041},
	{234.6168, 138.5512, 242.2665, 202.0349, 197.9338, 171.3064, 241.4041},
	{234.6168, 104.582, 242.2665, 166.0349, 197.9338, 173.0155, 205.9349},
	{202.1959, 104.582, 242.2665, 166.0349, 197.9338, 171.5155, 205.9349},
	{202.1959, 104.582, 207.2665, 99.5965, 197.9338, 171.5155, 206.9749},
	{202.1959, 104.582, 207.2665, 102.1365, 197.9338, 136.5155, 205.9349},
	{202.1959, 104.582, 207.2665, 100.9365, 197.9338, 136.5155, 206.5804},
	{202.1959, 104.582, 207.2665, 100.9365, 197.9338, 136.5155, 206.2659},
	{202.1959, 104.582, 207.2665, 100.9365, 196.8938, 134.83, 206.2659},
	{169.7267, 104.582, 207.2665, 100.9365, 198.5793, 136.33, 172.2967},
	{134.7267, 103.582, 207.2665, 100.9365, 166.1584, 136.33, 172.2967},
	{134.7267, 103.582, 207.2665, 100.9365, 166.1584, 135.33, 172.2967},
	{134.7267, 100.8965, 207.2665, 100.9365, 164.8284, 135.33, 172.2967},
	{134.7267, 100.8965, 204.2665, 100.9365, 197.2493, 135.33, 171.6667},
	{134.7267, 135.5657, 204.2665, 100.9365, 197.2493, 136.83, 204.0876},
	{134.7267, 135.8965, 204.2665, 100.9365, 197.2493, 136.83, 169.0876},
	{134.7267, 170.8965, 204.2665, 100.9365, 197.2493, 136.83, 135.1184},
	{134.7267, 170.8965, 204.2665, 100.9365, 197.2493, 137.4755, 135.1184},
	{100.7575, 170.8965, 203.2665, 100.9365, 197.2493, 172.46, 135.1184},
	{99.072, 169.8965, 201.7665, 100.9365, 164.8284, 173.96, 135.1184},
	{99.072, 169.8965, 201.7665, 100.9365, 164.8284, 173.96, 169.4184},
	{99.072, 169.8965, 201.7665, 100.9365, 164.8284, 172.92, 169.4184},
	{99.072, 169.8965, 201.7665, 100.9365, 164.8284, 174.6055, 169.4184},
	{99.072, 169.8965, 130.7665, 99.6065, 164.8284, 174.6055, 169.4184},
	{99.072, 169.8965, 130.7665, 130.9874, 164.8284, 174.6055, 167.9184},
	{99.072, 169.8965, 97.112, 134.0184, 164.8284, 174.6055, 167.9184},
	{99.072, 169.8965, 95.7665, 130.5429, 164.8284, 174.6055, 167.9184},
	{99.072, 169.8965, 132.2665, 165.1638, 163.1429, 174.6055, 167.9184},
	{99.072, 169.2665, 132.2665, 199.133, 128.1429, 139.6055, 167.9184},
	{98.072, 201.6874, 132.2665, 199.133, 128.1429, 141.291, 167.9184},
	{98.072, 200.0019, 164.0574, 199.133, 128.1429, 139.6055, 167.9184},
	{97.072, 198.6719, 164.0574, 199.133, 128.1429, 141.291, 167.9184},
	{97.072, 231.7928, 164.0574, 199.133, 131.352, 141.291, 167.9184},
	{97.072, 234.9783, 164.0574, 200.633, 131.352, 141.291, 135.4975},
	{97.072, 235.1638, 164.0574, 200.633, 131.352, 141.291, 169.4667},
	{97.072, 235.1638, 134.652, 198.433, 131.352, 140.491, 169.4667},
	{97.072, 234.8183, 168.6212, 199.433, 129.6665, 174.4602, 168.7667},
	{97.072, 234.8183, 168.6212, 199.433, 128.6665, 173.8302, 203.7667},
	{97.072, 234.8183, 168.6212, 199.433, 128.6665, 175.1602, 203.7667},
	{93.312, 234.8183, 168.6212, 199.433, 128.6665, 209.1294, 203.7667},
	{93.312, 234.8183, 167.9912, 199.433, 128.6665, 209.8294, 203.7667},
	{93.312, 199.8183, 200.4121, 199.433, 161.0874, 243.7986, 203.7667},
	{93.312, 163.8183, 200.4121, 199.433, 199.2649, 243.7986, 203.7667},
	{93.312, 162.3183, 232.833, 167.0121, 199.2649, 243.7986, 204.4667},
	{99.612, 162.3183, 232.833, 167.0121, 199.5957, 243.7986, 205.9667},
	{99.612, 162.3183, 232.833, 134.5912, 199.5957, 208.7986, 205.9667},
	{99.612, 161.6183, 232.833, 134.5912, 199.5957, 208.7986, 170.9667},
	{99.612, 129.1974, 232.493, 132.5912, 199.5957, 208.7986, 170.9667},
	{94.812, 129.1974, 234.1785, 133.2212, 199.5957, 208.7986, 170.9667},
	{92.042, 95.4365, 233.4785, 166.2049, 199.5957, 208.7986, 170.9667},
	{93.542, 97.122, 234.4785, 166.2049, 199.5957, 208.7986, 170.9667},
	{132.3112, 97.122, 234.4785, 130.5502, 199.5957, 208.7986, 170.9667},
	{132.3112, 97.122, 233.4385, 131.5357, 199.5957, 209.7986, 170.9667},
	{137.1112, 97.122, 200.124, 132.2357, 199.5957, 209.7986, 170.9667},
	{171.0804, 97.122, 200.124, 133.7357, 199.5957, 244.7986, 170.9667},
	{166.2804, 97.122, 235.124, 133.7357, 163.5957, 209.7986, 170.9667},
	{166.2804, 95.4365, 233.4385, 133.7357, 163.5957, 210.4986, 172.4667},
	{170.0804, 95.4365, 199.4693, 133.7357, 162.0957, 210.4986, 170.9667},
	{204.0496, 95.4365, 199.4693, 133.0357, 162.0957, 210.4986, 138.4975},
	{204.0496, 95.4365, 199.4693, 168.0357, 162.0957, 210.4986, 138.4975},
	{204.0496, 129.4057, 134.6275, 168.0357, 162.0957, 210.4986, 138.4975},
	{204.0496, 129.4057, 134.6275, 168.0357, 161.0957, 210.4986, 138.4975},
	{204.0496, 129.4057, 134.6275, 168.0357, 161.0957, 176.5294, 103.4975},
	{204.7496, 129.4057, 134.6275, 168.0357, 127.1265, 142.5602, 103.4975},
	{238.7188, 129.4057, 134.6275, 167.4057, 127.1265, 141.0602, 102.4975},
	{238.7188, 128.7757, 134.6275, 199.8266, 164.0965, 141.0602, 102.4975},
	{238.7188, 161.1966, 134.6275, 199.8266, 164.0965, 141.0602, 103.1975},
	{238.7188, 161.1966, 133.6275, 199.8266, 164.0965, 141.0602, 103.012},
	{238.7188, 161.1966, 133.6275, 199.8266, 164.0965, 141.0602, 103.012},
	{238.7188, 161.1966, 168.9267, 199.8266, 129.0965, 141.0602, 103.012},
	{238.7188, 160.1966, 168.9267, 199.8266, 129.0965, 141.0602, 103.012},
	{238.7188, 160.8966, 168.9267, 199.8266, 164.0965, 139.5602, 103.012},
	{237.7188, 162.3966, 168.9267, 199.8266, 129.0965, 139.5602, 103.012},
	{237.7188, 162.3966, 168.9267, 199.8266, 164.0965, 138.0602, 103.012},
	{169.7804, 162.0566, 168.9267, 165.8574, 164.0965, 138.0602, 103.712},
	{166.0204, 163.7421, 167.4267, 165.8574, 164.0965, 138.0602, 137.6812},
	{171.1204, 163.7421, 167.4267, 165.8574, 164.0965, 138.0602, 137.6812},
	{171.1204, 163.7421, 167.4267, 165.8574, 163.7565, 138.0602, 137.6812},
	{171.1204, 163.7421, 167.4267, 165.8574, 163.7565, 104.091, 137.6812},
	{171.1204, 163.7421, 132.4267, 165.8574, 163.7565, 104.391, 137.6812},
	{170.4904, 163.7421, 132.4267, 165.8574, 163.1265, 104.091, 170.1021},
	{168.9421, 162.2421, 132.4267, 165.8574, 197.2329, 105.591, 170.4021},
	{167.6121, 161.5421, 132.4267, 165.8574, 197.2329, 105.591, 169.0621},
	{200.033, 162.8721, 134.2667, 165.8574, 196.2329, 106.291, 170.7476},
	{200.033, 163.8721, 169.2667, 165.8574, 196.2329, 174.2294, 206.4168},
	{200.033, 163.5321, 169.2667, 133.4365, 196.2329, 174.2294, 206.4168},
	{200.033, 167.4176, 169.2667, 133.4365, 196.2329, 174.2294, 171.7476},
	{200.033, 167.4176, 169.2667, 98.4365, 196.2329, 173.5294, 206.7476},
	{200.3638, 135.3275, 169.2667, 98.4365, 196.2329, 207.4894, 209.2876},
	{200.3638, 167.7484, 169.2667, 98.4365, 196.2329, 209.1749, 209.2876},
	{200.3638, 167.7484, 169.2667, 98.4365, 161.2329, 209.1749, 209.2876},
	{200.3638, 165.5484, 170.2667, 98.4365, 162.7329, 209.8204, 208.5876},
	{200.3638, 166.5484, 205.5659, 98.4365, 162.7329, 209.8204, 243.5876},
	{200.3638, 166.5484, 170.2667, 98.4365, 162.7329, 207.1349, 243.5876},
	{200.3638, 166.5484, 204.0331, 164.8266, 161.0474, 208.8204, 243.5876},
	{200.3638, 198.9693, 237.6876, 133.7357, 161.0474, 208.8204, 243.5876},
	{200.3638, 198.9693, 237.0021, 167.7049, 161.3874, 243.1204, 209.6184},
	{200.3638, 200.3093, 239.3876, 167.7049, 127.3929, 208.1204, 209.6184},
	{200.3638, 200.3093, 240.8876, 167.7049, 129.0784, 208.1204, 177.1975},
	{200.3638, 200.3093, 240.8876, 167.7049, 129.0784, 208.1204, 175.6975},
	{164.5429, 200.3093, 242.3876, 167.7049, 96.012, 208.1204, 174.1975},
	{170.1429, 198.8093, 242.3876, 167.7049, 97.512, 242.7896, 174.1975},
	{171.1429, 198.8093, 242.3876, 167.7049, 96.512, 276.7588, 174.1975},
	{171.1429, 198.8093, 242.3876, 167.7049, 96.512, 276.7588, 174.1975},
	{133.922, 198.8093, 242.3876, 201.6741, 94.8265, 276.7588, 174.1975},
	{133.922, 198.8093, 242.3876, 201.6741, 94.8265, 242.7896, 174.1975},
	{132.2365, 198.8093, 242.3876, 201.6741, 95.5265, 241.7896, 173.1975},
	{135.7065, 197.1238, 207.3876, 203.8741, 98.0265, 241.7896, 171.6975},
	{168.1274, 197.1238, 205.7021, 203.8741, 98.0265, 207.8204, 171.6975},
	{168.1274, 197.1238, 205.7021, 205.5596, 96.6865, 207.8204, 171.6975},
	{168.1274, 165.4029, 205.7021, 203.0196, 98.372, 207.1204, 171.6975},
